		IF
			LEN(stMqttSettings.sMqttUserId) > 0
			AND LEN(stMqttSettings.sMqttPassword) > 0
		THEN
			iuLength := LEN(stMqttSettings.sMqttUserId)+2; (* 2 byte data length*)
			ipLength := LEN(stMqttSettings.sMqttPassword)+2; (* 2 byte data length*)
		ELSE
			iuLength := 0;
			ipLength := 0;
		END_IF

		(* Calculate length *)
		(* 10 byte header, 2 byte data length, data length, [user length + 2], [password length + 2]*)
		fbMqttEncodeLength(
			dwLength := 10 + 2 + INT_TO_BYTE(idLength) + INT_TO_BYTE(iuLength) + INT_TO_BYTE(ipLength),
			bLength1 => bLength1,
			bLength2 => bLength2,
			bLength3 => bLength3,
			bLength4 => bLength4,
			bAmount	 => bLengthAmount
		);

		(* MQTT Control Packet type *)
		stMqttTelegram.arMqttData[0] := 16;
		(* Remaining Length *)
		CASE bLengthAmount OF
			1:
				stMqttTelegram.arMqttData[1] := bLength1;

			2:
				stMqttTelegram.arMqttData[1] := bLength1;
				stMqttTelegram.arMqttData[2] := bLength2;

			3:
				stMqttTelegram.arMqttData[1] := bLength1;
				stMqttTelegram.arMqttData[2] := bLength2;
				stMqttTelegram.arMqttData[3] := bLength3;

			4:
				stMqttTelegram.arMqttData[1] := bLength1;
				stMqttTelegram.arMqttData[2] := bLength2;
				stMqttTelegram.arMqttData[3] := bLength3;
				stMqttTelegram.arMqttData[4] := bLength4;
		END_CASE;
		(* init position*)
		ipos := bLengthAmount;

		(* Length MSB *)
		stMqttTelegram.arMqttData[ipos+1] := 0;
		(* Length LSB *)
		stMqttTelegram.arMqttData[ipos+2] := 4;
		(* M *)
		stMqttTelegram.arMqttData[ipos+3] := 77;
		(* Q *)
		stMqttTelegram.arMqttData[ipos+4] := 81;
		(* T *)
		stMqttTelegram.arMqttData[ipos+5] := 84;
		(* T *)
		stMqttTelegram.arMqttData[ipos+6] := 84;
		(* Protocol Level *)
		stMqttTelegram.arMqttData[ipos+7] := 4;
		(* Connect Flags *)
		stMqttTelegram.arMqttData[ipos+8].1 := TRUE;
		stMqttTelegram.arMqttData[ipos+8].6 := (ipLength>2); (* more then 2 byte data length*)
		stMqttTelegram.arMqttData[ipos+8].7 := (iuLength>2); (* more then 2 byte data length*)
		(* Keep Alive MSB *)
		stMqttTelegram.arMqttData[ipos+9] := 0;
		(* Keep Alive LSB *)
		stMqttTelegram.arMqttData[ipos+10] := stMqttSettings.usKeepAliveTime;
		(* Data length MSB *)
		stMqttTelegram.arMqttData[ipos+11] := 0;
		(* Data length LSB *)
		stMqttTelegram.arMqttData[ipos+12] := INT_TO_BYTE(idLength);

		(* Client ID *)
		MEMCPY(
			destAddr	:= ADR(stMqttTelegram.arMqttData[ipos+13]),
		    srcAddr		:= ADR(stMqttSettings.sMqttClientId),
			n  			:= idLength
		);

		ipos := ipos+13+idLength;
		IF (iuLength > 2) THEN (* more then 2 byte data length*)
			(* Data length MSB *)
			stMqttTelegram.arMqttData[ipos] := 0;
			(* Data length LSB *)
			stMqttTelegram.arMqttData[ipos+1] := INT_TO_BYTE(iuLength-2);

			(* User ID *)
			MEMCPY(
				destAddr	:= ADR(stMqttTelegram.arMqttData[ipos+2]),
			    srcAddr		:= ADR(stMqttSettings.sMqttUserId),
				n  			:= iuLength-2
			);
			ipos := ipos+iuLength;
		END_IF

		IF (iuLength > 2) THEN (* more then 2 byte data length*)
			(* Data length MSB *)
			stMqttTelegram.arMqttData[ipos] := 0;
			(* Data length LSB *)
			stMqttTelegram.arMqttData[ipos+1] := INT_TO_BYTE(ipLength-2);

			(* Password *)
			MEMCPY(
				destAddr	:= ADR(stMqttTelegram.arMqttData[ipos+2]),
			    srcAddr		:= ADR(stMqttSettings.sMqttPassword),
				n  			:= ipLength-2
			);
			ipos := ipos+ipLength;
		END_IF

		stMqttTelegram.nDataLength 	:= ipos; (* 1 byte header, 1 byte remaining length *)
		iState 						:= C_SEND_WAIT;

	(* send telegram *)
	C_SEND_WAIT:
		IF stMqttSettings.stMqttSendTelegram.nDataLength = 0 THEN
			FC_Mqtt_CopyTelegram_V10(
				stMqttSrcTelegram	:= stMqttTelegram,
				stMqttDestTelegram	:= stMqttSettings.stMqttSendTelegram,
				stMqttSettings		:= stMqttSettings
			);

			stMqttSettings.bConnectPackageSent	:= TRUE;
			iState								:= C_IDLE;
		END_IF;

		IF
			NOT stMqttSettings.bActive
			OR NOT stMqttSettings.bSocketConnection
		THEN
			iState := C_STARTUP;
		END_IF;

	(* idle *)
	C_IDLE:
		IF
			NOT stMqttSettings.bDisconnect
			AND NOT stMqttSettings.bError
			AND NOT stMqttSettings.bConnected
			AND stMqttSettings.bSocketConnection
			AND NOT stMqttSettings.bConnectPackageSent
			AND stMqttSettings.bActive
		THEN
			iState := C_BUILD_CONNECT;
		END_IF;

		(* check received telegram *)
		IF
			stMqttSettings.bConnectPackageSent
			AND stMqttSettings.stMqttReceivedTelegram.nDataLength = 4
			AND stMqttSettings.stMqttReceivedTelegram.arMqttData[0] = 32
			AND stMqttSettings.stMqttReceivedTelegram.arMqttData[1] = 2
			AND (
				(* Session pressent or not, we ignore *)
				stMqttSettings.stMqttReceivedTelegram.arMqttData[2] = 1
				OR
				stMqttSettings.stMqttReceivedTelegram.arMqttData[2] = 0
			)
			AND stMqttSettings.stMqttReceivedTelegram.arMqttData[3] = 0
		THEN
			stMqttSettings.bConnected := TRUE;
			FC_Mqtt_ClearTelegram_V10(
				stMqttTelegram	:= stMqttSettings.stMqttReceivedTelegram,
				stMqttSettings	:= stMqttSettings
			);
		END_IF;

		(* error on connect *)
		IF
			stMqttSettings.bConnectPackageSent
			AND stMqttSettings.stMqttReceivedTelegram.nDataLength = 4
			AND stMqttSettings.stMqttReceivedTelegram.arMqttData[0] = 32
			AND stMqttSettings.stMqttReceivedTelegram.arMqttData[1] = 2
			AND stMqttSettings.stMqttReceivedTelegram.arMqttData[3] <> 0
		THEN
			stMqttSettings.bError := TRUE;
		END_IF;

		IF
			stMqttSettings.bDisconnect
			OR stMqttSettings.bError
			OR NOT stMqttSettings.bSocketConnection
			OR NOT stMqttSettings.bActive
		THEN
			iState := C_STARTUP;
		END_IF;

	ELSE
		iState := C_STARTUP;
END_CASE;


(*	END_FUNCTION_BLOCK	*)
END_FUNCTION_BLOCK

(* POU _Generic/Mqtt/Intern/FB_Mqtt_EncodeLength_V10, ST *)
FUNCTION_BLOCK FB_Mqtt_EncodeLength_V10
VAR_INPUT
	dwLength	: DWORD;
END_VAR
VAR_OUTPUT
	bLength1	: BYTE := 0;
	bLength2	: BYTE := 0;
	bLength3	: BYTE := 0;
	bLength4	: BYTE := 0;
	bAmount		: BYTE := 0;
END_VAR
VAR
	dwWorkLength	: DWORD;
	dwCopyLength	: DWORD;
END_VAR
(* @END_DECLARATION := '0' *)
bAmount 		:= 1;
dwCopyLength	:= dwLength;

WHILE dwCopyLength > 0 DO
	dwWorkLength := dwCopyLength MOD 128;
	dwCopyLength := dwCopyLength / 128;

	IF dwCopyLength > 0 THEN
		dwWorkLength := dwWorkLength OR 128;
	END_IF;

	CASE bAmount OF
		1:
			bLength1 := DWORD_TO_BYTE(dwWorkLength);

		2:
			bLength2 := DWORD_TO_BYTE(dwWorkLength);

		3:
			bLength3 := DWORD_TO_BYTE(dwWorkLength);

		4:
			bLength4 := DWORD_TO_BYTE(dwWorkLength);

		ELSE
			;
	END_CASE;

	IF dwCopyLength > 0 THEN
		bAmount := bAmount + 1;
	END_IF;

	IF bAmount > 4 THEN
		(* hmm *)
		RETURN;
	END_IF;
END_WHILE;
(*
do
	encodedByte = X MOD 128
	X = X DIV 128

	// if there are more data to encode, set the top bit of this byte
	if ( X > 0 )
		encodedByte = encodedByte OR 128
	endif

	'output' encodedByte
while ( X > 0 )
*)

(*	END_FUNCTION_BLOCK	*)
END_FUNCTION_BLOCK

(* POU _Generic/Mqtt/Intern/FC_Mqtt_ClearTelegram_V10, ST *)
FUNCTION FC_Mqtt_ClearTelegram_V10 : BOOL
VAR_IN_OUT
	stMqttTelegram	: ST_MqttTelegram;
	stMqttSettings	: ST_MqttSettings;
END_VAR
VAR
END_VAR
(* @END_DECLARATION := '0' *)
MEMSET(
	destAddr	:= ADR(stMqttTelegram.arMqttData),
	fillByte  	:= 0,
	n			:= stMqttSettings.iTelegramSize
);

stMqttTelegram.nDataLength := 0;

(*	END_FUNCTION	*)
END_FUNCTION

(* POU _Generic/Mqtt/Intern/FC_Mqtt_CopyTelegram_V10, ST *)
FUNCTION FC_Mqtt_CopyTelegram_V10 : BOOL
VAR_IN_OUT
	stMqttSrcTelegram	: ST_MqttTelegram;
	stMqttDestTelegram	: ST_MqttTelegram;
	stMqttSettings		: ST_MqttSettings;
END_VAR
VAR
END_VAR
(* @END_DECLARATION := '0' *)
MEMCPY(
	destAddr	:= ADR(stMqttDestTelegram.arMqttData),
    srcAddr		:= ADR(stMqttSrcTelegram.arMqttData),
	n  			:= stMqttSettings.iTelegramSize
);

stMqttDestTelegram.nDataLength := stMqttSrcTelegram.nDataLength;

(*	END_FUNCTION	*)
END_FUNCTION

(* POU _Generic/Mqtt/Intern/FB_MqttTelegram_PingReq_V10, ST *)
FUNCTION_BLOCK FB_MqttTelegram_PingReq_V10
VAR_IN_OUT
	stMqttSettings	: ST_MqttSettings;
END_VAR
VAR
	iState 				: INT := 0;
	bMustSend			: BOOL := FALSE;
	bPingReqSent		: BOOL := FALSE;
	stMqttTelegram		: ST_MqttTelegram;
END_VAR
VAR CONSTANT
	C_STARTUP		: INT := 0;
	C_BUILD_PING	: INT := 100;
	C_SEND_WAIT		: INT := 110;
	C_IDLE			: INT := 500;
END_VAR
(* @END_DECLARATION := '0' *)
CASE iState OF
	C_STARTUP:
		bPingReqSent := FALSE;

		IF stMqttSettings.bValidConnection THEN
			iState := C_IDLE;
		END_IF;

	(* build pingreq telegram *)
	C_BUILD_PING:
		FC_Mqtt_ClearTelegram_V10(
			stMqttTelegram	:= stMqttTelegram,
			stMqttSettings	:= stMqttSettings
		);

		(* MQTT Control Packet type *)
		stMqttTelegram.arMqttData[0] := 192;
		(* Remaining Length *)
		stMqttTelegram.arMqttData[1] := 0;

		stMqttTelegram.nDataLength := 2;

		iState := C_SEND_WAIT;

	(* send telegram *)
	C_SEND_WAIT:
		IF stMqttSettings.stMqttSendTelegram.nDataLength = 0 THEN
			FC_Mqtt_CopyTelegram_V10(
				stMqttSrcTelegram	:= stMqttTelegram,
				stMqttDestTelegram	:= stMqttSettings.stMqttSendTelegram,
				stMqttSettings		:= stMqttSettings
			);

			bPingReqSent	:= TRUE;
			iState			:= C_IDLE;
		END_IF;

		IF NOT stMqttSettings.bValidConnection THEN
			iState := C_STARTUP;
		END_IF;

	(* idle *)
	C_IDLE:
		bMustSend := FALSE;

		IF stMqttSettings.usKeepAliveTime > 0 THEN
			bMustSend := stMqttSettings.tonSendPingReq.Q;
		END_IF;

		IF
			stMqttSettings.bValidConnection
			AND bMustSend
			AND NOT bPingReqSent
		THEN
			iState := C_BUILD_PING;
		END_IF;

		(* Check received telegram *)
		IF
			bPingReqSent
			AND stMqttSettings.stMqttReceivedTelegram.nDataLength = 2
			AND stMqttSettings.stMqttReceivedTelegram.arMqttData[0] = 208
			AND stMqttSettings.stMqttReceivedTelegram.arMqttData[1] = 0
		THEN
			FC_Mqtt_ClearTelegram_V10(
				stMqttTelegram	:= stMqttSettings.stMqttReceivedTelegram,
				stMqttSettings	:= stMqttSettings
			);
			bPingReqSent := FALSE;
		END_IF;

		IF NOT stMqttSettings.bValidConnection THEN
			iState := C_STARTUP;
		END_IF;

	ELSE
		iState := C_STARTUP;
END_CASE;

(*	END_FUNCTION_BLOCK	*)
END_FUNCTION_BLOCK

(* POU _Generic/Mqtt/Intern/FB_Mqtt_Send_V10, ST *)
FUNCTION_BLOCK FB_Mqtt_Send_V10
VAR_OUTPUT
	bBusy	: BOOL := FALSE;
END_VAR
VAR_IN_OUT
	stMqttSettings	: ST_MqttSettings;
END_VAR
VAR
	fbSocketSend 	: FB_SocketSend;
	tPingReq		: TIME;
	iState 			: INT := 0;
	stSendTelegram	: ST_MqttTelegram;
END_VAR
VAR CONSTANT
	C_STARTUP		: INT := 0;
	C_SEND			: INT := 100;
	C_SEND_WAIT		: INT := 110;
	C_IDLE			: INT := 500;
END_VAR
(* @END_DECLARATION := '0' *)
CASE iState OF
	C_STARTUP:
		bBusy := FALSE;

		stMqttSettings.tonSendPingReq(
			in := FALSE
		);

		IF
			NOT stMqttSettings.bDisconnect
			AND NOT stMqttSettings.bError
			AND stMqttSettings.bSocketConnection
		THEN
			iState := C_IDLE;
		END_IF;

	(* send mqtt telegram *)
	C_SEND:
		bBusy := TRUE;

		(* copy send telegram *)
		FC_Mqtt_CopyTelegram_V10(
			stMqttSrcTelegram	:= stMqttSettings.stMqttSendTelegram,
			stMqttDestTelegram	:= stSendTelegram,
			stMqttSettings		:= stMqttSettings
		);

		(* start send *)
		fbSocketSend(
			bExecute := FALSE
		);

		fbSocketSend(
			sSrvNetId	:= '',
			hSocket		:= stMqttSettings.hSocket,
			cbLen		:= stSendTelegram.nDataLength,
			pSrc		:= ADR(stSendTelegram.arMqttData),
			bExecute 	:= TRUE
		);

		iState := C_SEND_WAIT;

	(* wait send done *)
	C_SEND_WAIT:
		fbSocketSend(
			bExecute := FALSE
		);

		IF
			NOT fbSocketSend.bBusy
			AND NOT fbSocketSend.bError
		THEN
			(* copy last telegram *)
			FC_Mqtt_CopyTelegram_V10(
				stMqttSrcTelegram	:= stMqttSettings.stMqttSendTelegram,
				stMqttDestTelegram	:= stMqttSettings.stMqttLastSendTelegram,
				stMqttSettings		:= stMqttSettings
			);

			(* clear send buffer *)
			FC_Mqtt_ClearTelegram_V10(
				stMqttTelegram 	:= stMqttSettings.stMqttSendTelegram,
				stMqttSettings	:= stMqttSettings
			);

			iState	:= C_IDLE;
			bBusy	:= FALSE;
		END_IF;

		IF stMqttSettings.usKeepAliveTime > 0 THEN
			tPingReq := DWORD_TO_TIME(USINT_TO_DWORD(stMqttSettings.usKeepAliveTime) * 1000 - 5000);

			stMqttSettings.tonSendPingReq(
				in := FALSE
			);

			stMqttSettings.tonSendPingReq(
				in := TRUE,
				pt := tPingReq
			);
		END_IF;

		IF fbSocketSend.bError THEN
			iState 					:= C_STARTUP;
			stMqttSettings.bError	:= TRUE;
		END_IF;

		IF
			NOT stMqttSettings.bActive
			OR NOT stMqttSettings.bSocketConnection
		THEN
			iState := C_STARTUP;
		END_IF;

	(* idle *)
	C_IDLE:
		IF stMqttSettings.usKeepAliveTime > 0 THEN
			stMqttSettings.tonSendPingReq(
				in := stMqttSettings.bConnected
			);
		ELSE
			stMqttSettings.tonSendPingReq(
				in := FALSE
			);
		END_IF;

		IF
			stMqttSettings.stMqttSendTelegram.nDataLength > 0
			AND NOT stMqttSettings.bDisconnect
			AND NOT stMqttSettings.bError
			AND stMqttSettings.bSocketConnection
			AND NOT bBusy
		THEN
			iState := C_SEND;
		END_IF;

		IF
			stMqttSettings.bDisconnect
			OR stMqttSettings.bError
			OR NOT stMqttSettings.bSocketConnection
		THEN
			iState := C_STARTUP;
		END_IF;

		(* ensure at least 1 cycle pause *)
		(* bBusy := FALSE; *)

	ELSE
		iState := C_STARTUP;
END_CASE;

(*	END_FUNCTION_BLOCK	*)
END_FUNCTION_BLOCK

(* POU _Generic/Mqtt/Intern/FB_Mqtt_Receive_V10, ST *)
FUNCTION_BLOCK FB_Mqtt_Receive_V10
VAR_OUTPUT
	bBusy	: BOOL := FALSE;
END_VAR
VAR_IN_OUT
	stMqttSettings	: ST_MqttSettings;
END_VAR
VAR
	fbSocketReceive		: FB_SocketReceive;
	fbMqttDecodeLength	: FB_Mqtt_DecodeLength_V10;
	stReceiveBuffer		: ST_MqttTelegram;

	iState 			: INT := 0;
	iLengthPosition	: INT := 0;
	index			: INT := 0;
	dwDataLength	: DWORD := 0;
	wTopicLength	: WORD := 0;
	dwValueLength	: DWORD := 0;
END_VAR
VAR CONSTANT
	C_STARTUP				: INT := 0;
	C_RECEIVE_HEADER		: INT := 100;
	C_RECEIVE_HEADER_WAIT	: INT := 110;
	C_RECEIVE_LENGTH		: INT := 120;
	C_RECEIVE_LENGTH_WAIT	: INT := 130;
	C_RECEIVE_DATA			: INT := 200;
	C_RECEIVE_DATA_WAIT		: INT := 210;
	C_IDLE					: INT := 500;
END_VAR
(* @END_DECLARATION := '0' *)
CASE iState OF
	C_STARTUP:
		bBusy 			:= FALSE;
		iLengthPosition	:= 0;
		index			:= 0;
		dwDataLength	:= 0;
		wTopicLength	:= 0;
		dwValueLength	:= 0;
		ClearReceivedPublishTelegram();

		IF
			NOT stMqttSettings.bDisconnect
			AND NOT stMqttSettings.bError
			AND stMqttSettings.bSocketConnection
		THEN
			iState := C_IDLE;
		END_IF;

	(* start receive header *)
	C_RECEIVE_HEADER:
		bBusy := TRUE;
		ClearReceivedPublishTelegram();

		fbSocketReceive(
			bExecute := FALSE
		);

		fbSocketReceive(
			sSrvNetId	:= '',
			hSocket		:= stMqttSettings.hSocket,
			cbLen		:= 2,
			pDest		:= ADR(stReceiveBuffer.arMqttData),
			bExecute 	:= TRUE
		);

		iState := C_RECEIVE_HEADER_WAIT;

	(* wait for header with length *)
	C_RECEIVE_HEADER_WAIT:
		fbSocketReceive(
			bExecute := FALSE
		);

		IF
			NOT fbSocketReceive.bBusy
			AND NOT fbSocketReceive.bError
			AND fbSocketReceive.nRecBytes = 2
		THEN
			iLengthPosition	:= 0;
			stMqttSettings.stMqttReceivedTelegram.arMqttData[0] := stReceiveBuffer.arMqttData[0];
			stMqttSettings.stMqttReceivedTelegram.arMqttData[1] := stReceiveBuffer.arMqttData[1];

			IF stMqttSettings.stMqttReceivedTelegram.arMqttData[1].7 = 1 THEN
				(* payload longer then 127 byte *)
				iLengthPosition := iLengthPosition + 1;
				iState			:= C_RECEIVE_LENGTH;
			ELSE
				IF stMqttSettings.stMqttReceivedTelegram.arMqttData[1] = 0 THEN
					(* no payload received *)
					stMqttSettings.stMqttReceivedTelegram.nDataLength := 2;

					(* copy last telegram *)
					FC_Mqtt_CopyTelegram_V10(
						stMqttSrcTelegram	:= stMqttSettings.stMqttReceivedTelegram,
						stMqttDestTelegram	:= stMqttSettings.stMqttLastReceivedTelegram,
						stMqttSettings		:= stMqttSettings
					);

					iState	:= C_IDLE;
					bBusy 	:= FALSE;
				ELSE
					iState := C_RECEIVE_DATA;
				END_IF;
			END_IF;
		END_IF;

		IF fbSocketReceive.bError THEN
			iState 					:= C_STARTUP;
			stMqttSettings.bError	:= TRUE;
		END_IF;

		IF fbSocketReceive.nRecBytes = 0 THEN
			iState	:= C_IDLE;
			bBusy	:= FALSE;
		END_IF;

		IF
			NOT stMqttSettings.bActive
			OR NOT stMqttSettings.bSocketConnection
		THEN
			iState := C_STARTUP;
		END_IF;

	(* read next remaining length *)
	C_RECEIVE_LENGTH:
		fbSocketReceive(
			bExecute := FALSE
		);

		fbSocketReceive(
			sSrvNetId	:= '',
			hSocket		:= stMqttSettings.hSocket,
			cbLen		:= 1,
			pDest		:= ADR(stReceiveBuffer.arMqttData),
			bExecute 	:= TRUE
		);

		iState := C_RECEIVE_LENGTH_WAIT;

	(* wait for remaining length *)
	C_RECEIVE_LENGTH_WAIT:
		fbSocketReceive(
			bExecute := FALSE
		);

		IF
			NOT fbSocketReceive.bBusy
			AND NOT fbSocketReceive.bError
			AND fbSocketReceive.nRecBytes = 1
		THEN
			stMqttSettings.stMqttReceivedTelegram.arMqttData[1 + iLengthPosition] := stReceiveBuffer.arMqttData[0];

			IF stMqttSettings.stMqttReceivedTelegram.arMqttData[1 + iLengthPosition].7 = 1 THEN
				(* read next length byte *)
				iLengthPosition := iLengthPosition + 1;
				iState			:= C_RECEIVE_LENGTH;

				(* Not more the 4 length bytes *)
				IF iLengthPosition > 4 THEN
					iState 					:= C_STARTUP;
					stMqttSettings.bError	:= TRUE;
				END_IF;
			ELSE
				iState := C_RECEIVE_DATA;
			END_IF;
		END_IF;

		IF fbSocketReceive.bError THEN
			iState 					:= C_STARTUP;
			stMqttSettings.bError	:= TRUE;
		END_IF;

		IF
			NOT stMqttSettings.bActive
			OR NOT stMqttSettings.bSocketConnection
		THEN
			iState := C_STARTUP;
		END_IF;

	(* receive remaining data *)
	C_RECEIVE_DATA:
		fbMqttDecodeLength(
			stMqttTelegram	:= stMqttSettings.stMqttReceivedTelegram,
			dwLength		=> dwDataLength
		);

		fbSocketReceive(
			bExecute := FALSE
		);

		fbSocketReceive(
			sSrvNetId	:= '',
			hSocket		:= stMqttSettings.hSocket,
			cbLen		:= dwDataLength,
			pDest		:= ADR(stReceiveBuffer.arMqttData),
			bExecute 	:= TRUE
		);

		iState := C_RECEIVE_DATA_WAIT;

	(* receive *)
	C_RECEIVE_DATA_WAIT:
		fbSocketReceive(
			bExecute := FALSE
		);

		IF
			NOT fbSocketReceive.bBusy
			AND NOT fbSocketReceive.bError
			AND fbSocketReceive.nRecBytes > 0
		THEN
			MEMCPY(
				destAddr	:= ADR(stMqttSettings.stMqttReceivedTelegram.arMqttData[2 + iLengthPosition]),
			    srcAddr		:= ADR(stReceiveBuffer.arMqttData),
				n  			:= fbSocketReceive.nRecBytes
			);
			stMqttSettings.stMqttReceivedTelegram.nDataLength := 2 + iLengthPosition + fbSocketReceive.nRecBytes;

			(* copy last telegram *)
			FC_Mqtt_CopyTelegram_V10(
				stMqttSrcTelegram	:= stMqttSettings.stMqttReceivedTelegram,
				stMqttDestTelegram	:= stMqttSettings.stMqttLastReceivedTelegram,
				stMqttSettings		:= stMqttSettings
			);

			(* check for publish *)
			IF (stMqttSettings.stMqttReceivedTelegram.arMqttData[0] AND 48) = 48 THEN
				ClearReceivedPublishTelegram();

				(* Length MSB/LSB Topic *)
				wTopicLength :=
						SHL(BYTE_TO_WORD(stMqttSettings.stMqttReceivedTelegram.arMqttData[2 + iLengthPosition + 1]), 8) +
						BYTE_TO_WORD(stMqttSettings.stMqttReceivedTelegram.arMqttData[1 + iLengthPosition + 1]);
				wTopicLength := BE16_TO_HOST(wTopicLength);

				(* Copy topic *)
				MEMCPY(
					destAddr	:= ADR(stMqttSettings.stMqttReceivedPublishTelegram.sTopic),
				    srcAddr		:= ADR(stMqttSettings.stMqttReceivedTelegram.arMqttData[3 + iLengthPosition + 1]),
					n  			:= wTopicLength
				);

				(* Copy value *)
				(* value length = remaining data length - length topic value - 2 byte topic length *)
				dwValueLength := dwDataLength - wTopicLength - 2;

				MEMCPY(
					destAddr	:= ADR(stMqttSettings.stMqttReceivedPublishTelegram.sValue),
				    srcAddr		:= ADR(stMqttSettings.stMqttReceivedTelegram.arMqttData[3 + iLengthPosition + 1 + wTopicLength]),
					n  			:= dwValueLength
				);

				stMqttSettings.stMqttReceivedPublishTelegram.bHasData := TRUE;
			END_IF;

			iState	:= C_IDLE;
			bBusy	:= FALSE;
		END_IF;

		IF fbSocketReceive.bError THEN
			iState 					:= C_STARTUP;
			stMqttSettings.bError	:= TRUE;
		END_IF;

		IF
			NOT stMqttSettings.bActive
			OR NOT stMqttSettings.bSocketConnection
		THEN
			iState := C_STARTUP;
		END_IF;

	(* idle *)
	C_IDLE:
		IF
			NOT stMqttSettings.bDisconnect
			AND NOT stMqttSettings.bError
			AND stMqttSettings.bSocketConnection
			AND NOT bBusy
		THEN
			iState := C_RECEIVE_HEADER;
		END_IF;

		IF
			stMqttSettings.bDisconnect
			OR stMqttSettings.bError
			OR NOT stMqttSettings.bSocketConnection
		THEN
			iState := C_STARTUP;
		END_IF;

		(* ensure at least 1 cycle pause *)
		(* bBusy := FALSE; *)

	ELSE
		iState := C_STARTUP;
END_CASE;

(*	END_FUNCTION_BLOCK	*)
END_FUNCTION_BLOCK
ACTION ClearReceivedPublishTelegram:
MEMSET(
	destAddr	:= ADR(stMqttSettings.stMqttReceivedPublishTelegram.sTopic),
	fillByte  	:= 0,
	n			:= 255
);
stMqttSettings.stMqttReceivedPublishTelegram.sTopic := '';

MEMSET(
	destAddr	:= ADR(stMqttSettings.stMqttReceivedPublishTelegram.sValue),
	fillByte  	:= 0,
	n			:= 255
);
stMqttSettings.stMqttReceivedPublishTelegram.sValue := '';

stMqttSettings.stMqttReceivedPublishTelegram.bHasData := FALSE;
END_ACTION

(* POU _Generic/Mqtt/Intern/FB_Mqtt_DecodeLength_V10, ST *)
FUNCTION_BLOCK FB_Mqtt_DecodeLength_V10
VAR_INPUT
	stMqttTelegram : ST_MqttTelegram;
END_VAR
VAR_OUTPUT
	dwLength	: DWORD;
	bAmount		: BYTE;
END_VAR
VAR
	index			: INT;
	diMultiplier	: DINT;
	dwValue			: DWORD;
END_VAR
(* @END_DECLARATION := '0' *)
index			:= 0;
diMultiplier	:= 1;
dwValue			:= 0;

REPEAT
	index := index + 1;

	dwValue := dwValue + (stMqttTelegram.arMqttData[index] AND 127) * diMultiplier;
	diMultiplier := diMultiplier * 128;

	IF diMultiplier > 128*128*128 THEN
		dwLength	:= 0;
		bAmount		:= 0;
		RETURN;
	END_IF;
UNTIL stMqttTelegram.arMqttData[index].7 = 0
END_REPEAT;

dwLength	:= dwValue;
bAmount		:= INT_TO_BYTE(index);

(*
multiplier = 1
value = 0

do
	encodedByte = 'next byte from stream'
	value += (encodedByte AND 127) * multiplier
	multiplier *= 128

	if (multiplier > 128*128*128)
		throw Error(Malformed Remaining Length)
while ((encodedByte AND 128) != 0)

*)

(*	END_FUNCTION_BLOCK	*)
END_FUNCTION_BLOCK

(* POU _Generic/Mqtt/FB_Mqtt_Publish_V10, ST *)
FUNCTION_BLOCK FB_Mqtt_Publish_V10
VAR_INPUT
	sTopic	: STRING[255];
	sValue	: STRING[255];
	bRetain	: BOOL := TRUE;
END_VAR
VAR_OUTPUT
	bBusy	: BOOL := FALSE;
END_VAR
VAR_IN_OUT
	stMqttSettings	: ST_MqttSettings;
END_VAR
VAR
	bFirstPublishDone	: BOOL := FALSE;
	bMustPublish		: BOOL := FALSE;
	sLastValue			: STRING[255];
	iState 				: INT := 0;
	iLengthTopic		: INT := 0;
	iLengthValue		: INT := 0;
	wTopicLength		: WORD;
	stMqttTelegram		: ST_MqttTelegram;
	fbMqttEncodeLength	: FB_Mqtt_EncodeLength_V10;
	bLength1			: BYTE;
	bLength2			: BYTE;
	bLength3			: BYTE;
	bLength4			: BYTE;
	bLengthAmount		: BYTE;
END_VAR
VAR CONSTANT
	C_STARTUP			: INT := 0;
	C_BUILD_TELEGRAM	: INT := 100;
	C_SEND_WAIT			: INT := 110;
	C_IDLE				: INT := 500;
END_VAR
(* @END_DECLARATION := '0' *)
CASE iState OF
	C_STARTUP:
		bFirstPublishDone	:= FALSE;
		bBusy				:= FALSE;

		IF stMqttSettings.bValidConnection THEN
			iState := C_IDLE;
		END_IF;

	(* build publish telegram *)
	C_BUILD_TELEGRAM:
		bBusy := TRUE;
		iLengthTopic := LEN(sTopic);
		iLengthValue := LEN(sValue);

		FC_Mqtt_ClearTelegram_V10(
			stMqttTelegram	:= stMqttTelegram,
			stMqttSettings	:= stMqttSettings
		);

		wTopicLength := iLengthTopic;
		wTopicLength := HOST_TO_BE16(wTopicLength);

		(* Calculate length *)
		(* 2 byte length topic, x byte length topic, x byte length value *)
		fbMqttEncodeLength(
			dwLength := 2 + iLengthTopic + iLengthValue,
			bLength1 => bLength1,
			bLength2 => bLength2,
			bLength3 => bLength3,
			bLength4 => bLength4,
			bAmount	 => bLengthAmount
		);

		(* MQTT Control Packet type, no DUP, no QoS, Retain *)
		stMqttTelegram.arMqttData[0] := 48;
		IF bRetain THEN
			stMqttTelegram.arMqttData[0].0 := 1;
		END_IF;

		(* Remaining Length *)
		CASE bLengthAmount OF
			1:
				stMqttTelegram.arMqttData[1] := bLength1;

			2:
				stMqttTelegram.arMqttData[1] := bLength1;
				stMqttTelegram.arMqttData[2] := bLength2;

			3:
				stMqttTelegram.arMqttData[1] := bLength1;
				stMqttTelegram.arMqttData[2] := bLength2;
				stMqttTelegram.arMqttData[3] := bLength3;

			4:
				stMqttTelegram.arMqttData[1] := bLength1;
				stMqttTelegram.arMqttData[2] := bLength2;
				stMqttTelegram.arMqttData[3] := bLength3;
				stMqttTelegram.arMqttData[4] := bLength4;

			ELSE
				iState 					:= C_STARTUP;
				stMqttSettings.bError	:= TRUE;
		END_CASE;

		(* Length MSB Topic *)
		stMqttTelegram.arMqttData[1 + bLengthAmount] := WORD_TO_BYTE(wTopicLength);
		(* Length LSB Topic *)
		stMqttTelegram.arMqttData[2 + bLengthAmount] := WORD_TO_BYTE(SHR(wTopicLength, 8));

		(* Add topic *)
		MEMCPY(
			destAddr	:= ADR(stMqttTelegram.arMqttData[3 + bLengthAmount]),
		    srcAddr		:= ADR(sTopic),
			n  			:= iLengthTopic
		);

		(* Add Payload *)
		MEMCPY(
			destAddr	:= ADR(stMqttTelegram.arMqttData[3 + bLengthAmount + iLengthTopic]),
		    srcAddr		:= ADR(sValue),
			n  			:= iLengthValue
		);

		(* 1 byte header, x byte variable length, 2 byte topic lenght, x byte topic, x byte value *)
		stMqttTelegram.nDataLength := 1 + bLengthAmount + 2 + iLengthTopic + iLengthValue;

		iState := C_SEND_WAIT;

	(* send telegram *)
	C_SEND_WAIT:
		IF stMqttSettings.stMqttSendTelegram.nDataLength = 0 THEN
			FC_Mqtt_CopyTelegram_V10(
				stMqttSrcTelegram	:= stMqttTelegram,
				stMqttDestTelegram	:= stMqttSettings.stMqttSendTelegram,
				stMqttSettings		:= stMqttSettings
			);

			iState				:= C_IDLE;
			bFirstPublishDone	:= TRUE;
			sLastValue			:= sValue;
		END_IF;

		IF NOT stMqttSettings.bValidConnection THEN
			iState := C_STARTUP;
		END_IF;

	(* idle *)
	C_IDLE:
		bBusy 			:= FALSE;
		bMustPublish 	:= sLastValue <> sValue;

		IF
			stMqttSettings.bValidConnection
			AND (
				bMustPublish
				OR NOT bFirstPublishDone
			)
		THEN
			iState := C_BUILD_TELEGRAM;
		END_IF;

		IF NOT stMqttSettings.bValidConnection THEN
			iState := C_STARTUP;
		END_IF;

	ELSE
		iState := C_STARTUP;
END_CASE;

(*	END_FUNCTION_BLOCK	*)
END_FUNCTION_BLOCK

(* POU ParnikWindowCtrl_old, ST *)
PROGRAM ParnikWindowCtrl_old
VAR
    (* Modbus I/O (использовать точно как заданы) *)
    (* Modbus.Street_temp : REAL *)
    (* Modbus.Parnik_set_temp_street_min : REAL *)
    (* Modbus.Parnik_air_temp : REAL *)
    (* Modbus.Parnik_set_auto_window : BOOL *)
    (* Modbus.Parnik_current_level_window : UINT *) (* 0=closed,1=30%,2=60%,3=100% *)
    (* Modbus.Parnik_manual_level_window : UINT *)
    (* Modbus.Parnik_temp_step1_window : UINT *) (* threshold for 30% *)
    (* Modbus.Parnik_temp_step2_window : UINT *) (* threshold for 60% *)

    (* HW outputs *)
    (* HW_power_supply_parnik : BOOL *)
    (* HW_power_polarity_parnik : BOOL *)

    (* Internal *)
    closeTON : TON;                 (* PT = 60s *)
    openTON  : TON;                 (* PT = variable *)
    state : UINT := 0;              (* 0=idle,1=closing,2=opening *)
    targetLevel : UINT := 0;        (* desired final level 0..3 *)
    openTime : TIME := T#0s;
    hysteresis : REAL := 4.0;
    prevManualLevel : UINT := 255;
    manualReq : BOOL := FALSE;
    startClose : BOOL := FALSE;
    startOpen  : BOOL := FALSE;
    firstScan : BOOL := TRUE;
END_VAR
IF firstScan THEN
    Modbus.Parnik_current_level_window := 0; (* default closed *)
    HW_power_supply_parnik := FALSE;
    HW_power_polarity_parnik := FALSE;
    closeTON(IN := FALSE, PT := T#60s);
    openTON(IN := FALSE, PT := T#60s);
    prevManualLevel := Modbus.Parnik_manual_level_window;
    firstScan := FALSE;
END_IF

(* detect manual change request *)
manualReq := FALSE;
IF NOT Modbus.Parnik_set_auto_window THEN
    IF Modbus.Parnik_manual_level_window <> prevManualLevel THEN
        manualReq := TRUE;
    END_IF;
END_IF;
prevManualLevel := Modbus.Parnik_manual_level_window;

(* Determine targetLevel according to requested logic *)
IF Modbus.Parnik_set_auto_window THEN
    (* AUTO *)
    IF (Modbus.Parnik_air_temp > (INT_TO_REAL(Modbus.Parnik_temp_step1_window) + hysteresis))
       AND (Modbus.Parnik_air_temp < INT_TO_REAL(Modbus.Parnik_temp_step2_window))
       AND (Modbus.Street_temp > Modbus.Parnik_set_temp_street_min) THEN
        targetLevel := 1; (* 30% *)
    ELSIF (Modbus.Parnik_air_temp > (INT_TO_REAL(Modbus.Parnik_temp_step2_window) + hysteresis))
       AND (Modbus.Street_temp > Modbus.Parnik_set_temp_street_min) THEN
        targetLevel := 2; (* 60% *)
    ELSIF ( (Modbus.Parnik_air_temp < (INT_TO_REAL(Modbus.Parnik_temp_step1_window) - hysteresis))
            OR (Modbus.Street_temp < Modbus.Parnik_set_temp_street_min) ) THEN
        targetLevel := 0; (* close *)
    ELSE
        targetLevel := Modbus.Parnik_current_level_window; (* keep current *)
    END_IF;
ELSE
    (* MANUAL - independent от температуры *)
    CASE Modbus.Parnik_manual_level_window OF
        0: targetLevel := 0;
        1: targetLevel := 1;
        2: targetLevel := 2;
        3: targetLevel := 3;
        ELSE targetLevel := Modbus.Parnik_current_level_window;
    END_CASE;
END_IF;


(* Helper: request sequence when target differs or when manualReq *)
IF state = 0 THEN
    startClose := FALSE;
    startOpen := FALSE;
    (* If target equals current -> nothing *)
    IF Modbus.Parnik_current_level_window <> targetLevel THEN
        IF targetLevel = 0 THEN
            (* need close *)
            startClose := TRUE;
            state := 1;
            HW_power_polarity_parnik := FALSE; (* closing polarity *)
        ELSE
            (* target > 0 *)
            IF Modbus.Parnik_current_level_window < targetLevel THEN
                (* already closed -> open directly *)
(*                IF openTime > T#0s THEN *)
                    startOpen := TRUE;
			IF (Modbus.Parnik_current_level_window = 0 AND targetLevel  = 1) THEN
		 	   openTime := T#5s;
			 END_IF
			IF (Modbus.Parnik_current_level_window = 0 AND targetLevel =  2) THEN
		 	   openTime := T#30s;
			 END_IF
			IF (Modbus.Parnik_current_level_window = 0 AND targetLevel =  3) THEN
		 	   openTime := T#60s;
			 END_IF
			IF (Modbus.Parnik_current_level_window = 1 AND targetLevel =  2) THEN
		 	   openTime := T#20s;
			 END_IF
			IF (Modbus.Parnik_current_level_window = 1 AND targetLevel =  3) THEN
		 	   openTime := T#50s;
			 END_IF
			IF (Modbus.Parnik_current_level_window = 2 AND targetLevel =  3) THEN
		 	   openTime := T#30s;
			 END_IF
                    state := 2;
                    HW_power_polarity_parnik := TRUE; (* opening polarity *)
            ELSE
                (* not closed -> close first *)
                startClose := TRUE;
                state := 1;
                HW_power_polarity_parnik := FALSE;
            END_IF;
        END_IF;
    END_IF;
END_IF

(* Also handle explicit manual request forcing sequence even if target==current but user changed set *)
IF manualReq AND (state = 0) THEN
    IF Modbus.Parnik_current_level_window <> targetLevel THEN
        (* same logic as above: if target>0 and already closed -> open; else close first *)
        IF targetLevel = 0 THEN
            startClose := TRUE; state := 1; HW_power_polarity_parnik := FALSE;
        ELSE
            IF Modbus.Parnik_current_level_window = 0 THEN
                IF openTime > T#0s THEN startOpen := TRUE; state := 2; HW_power_polarity_parnik := TRUE;
                ELSE Modbus.Parnik_current_level_window := targetLevel; state := 0;
                END_IF;
            ELSE
                startClose := TRUE; state := 1; HW_power_polarity_parnik := FALSE;
            END_IF;
        END_IF;
    END_IF;
END_IF

(* State machine with explicit TON IN handling *)
CASE state OF
    0: (* idle *)
        HW_power_supply_parnik := FALSE;
    1: (* closing - use full close time 60s *)
        closeTON(IN := startClose, PT := T#60s);
        HW_power_polarity_parnik := FALSE;
        HW_power_supply_parnik := startClose;

        IF closeTON.Q THEN
            (* finished closing *)
            closeTON(IN := FALSE, PT := T#60s);
            startClose := FALSE;
            HW_power_supply_parnik := FALSE;
            Modbus.Parnik_current_level_window := 0;
            (* If target >0 -> open to required level *)
            IF targetLevel > 0 THEN
                IF openTime > T#0s THEN
                    startOpen := TRUE;
                    state := 2;
                    HW_power_polarity_parnik := TRUE;
                ELSE
                    Modbus.Parnik_current_level_window := targetLevel;
                    state := 0;
                END_IF;
            ELSE
                state := 0;
            END_IF;
        END_IF;

    2: (* opening *)
        IF openTime = T#0s THEN
            startOpen := FALSE;
            HW_power_supply_parnik := FALSE;
            Modbus.Parnik_current_level_window := targetLevel;
            state := 0;
        ELSE
            openTON(IN := startOpen, PT := openTime);
            HW_power_polarity_parnik := TRUE;
            HW_power_supply_parnik := startOpen;

            IF openTON.Q THEN
                openTON(IN := FALSE, PT := openTime);
                startOpen := FALSE;
                HW_power_supply_parnik := FALSE;
                Modbus.Parnik_current_level_window := targetLevel;
                state := 0;
            END_IF;
        END_IF;

ELSE
    (* fallback safe *)
    HW_power_supply_parnik := FALSE;
    startClose := FALSE;
    startOpen := FALSE;
    closeTON(IN := FALSE, PT := T#60s);
    openTON(IN := FALSE, PT := openTime);
    state := 0;
END_CASE;
END_PROGRAM

(* POU RS485read_2_old, ST *)
PROGRAM RS485read_2_old
VAR
	password_1				: ARRAY [1..6] OF BYTE:=6(1); (* пароль к меркуриям, по умолчанию 6 единиц*)






	get_energy_E_T1			: FB_GET_ENERGY;
	get_energy_E_T2			: FB_GET_ENERGY;
	get_energy_MT			: FB_GET_ENERGY;
	get_supply				: FB_GET_SUPPLY;
	get_current				: FB_GET_CURRENT;
	get_power				: FB_GET_POWER;
	energyMT					: ARRAY[1..12,1..2] OF REAL;

	get_current_done			: BOOL;
	get_power_done			: BOOL;

	get_energy_E_T1_done	: BOOL;
	get_energy_E_T2_done	: BOOL;
	get_energy_MT_done		: BOOL;

	get_supply_done			: BOOL;
(*	CounterError_M			: DINT;
	CounterSuccess_M		: DINT;
*)




	flag: BOOL := TRUE;
	KLConfiguration: KL6configuration;
(*	Period_vent_switch	: INT:=180; *)
	CO2_period			: TIME;
	tTimerValue			: TIME	:=	t#10s; (* Период опроса RS485*)

	crctest					: WORD;

	arrReceive				: ARRAY[1..5] OF BYTE;
	arrSend					: ARRAY[1..5] OF BYTE;

	MBdata					 : ARRAY [1..2] OF INT;
	MBdata_pzem			 : ARRAY [1..2] OF INT;
	MBdata8					 : ARRAY [1..8] OF INT;
	FtrigBusy				: F_TRIG;
	timeoutvalue				: TIME := T#2000ms;		(* timeout while waiting for an answer of the modbus slave *)
	state					: INT;
	busy					: BOOL;
	LastErrorstate				: INT;
	LastModbusError			: ST_ModbusErrorDiagnostics;
	CounterError				: DINT;
	CounterSuccess			: DINT;

	i,k,l,m,t					: INT:=1;



	sensors_CO2_id				: ARRAY[1..2] OF BYTE:=16#68, 16#69;
	sensors_CO2_ppm			: ARRAY[1..2] OF INT;

	sensors_PZEM_id			: BYTE:=16#02;
	sensors_PZEM_data		: ARRAY[1..2] OF REAL:=2(0);

	sensors_DS18B20_id			: BYTE:=16#01;
	sensors_DS18B20_temp		: ARRAY[1..8] OF REAL:=8(0);


	get_co2_mh_z19b_1floor	: FB_GET_CO2_MH_Z19B;
(*	get_co2_mh_z19b_2floor	: FB_GET_CO2_MH_Z19B; *)
	get_co2_mh_z19b_1floor_done	: BOOL;
(*	get_co2_mh_z19b_2floor_done	: BOOL; *)
	sensor_ponics_PH_id		: BYTE:= 16#4F ;
	MBdata_sensor_ponics_PH : ARRAY [1..4] OF INT;
	Ponics_PH_temp			: REAL;

	sensor_ponics_PH_int		:INT;

	sensor_ponics_EC_id		: BYTE:= 16#51 ;
(*	sensor_ponics_EC2_id		: BYTE:= 16#50 ; *)
	sensor_ponics_EC_int		:INT;

	balkon_light_sensor_id			: BYTE:=16#5A;
	balkon_light_low				: BYTE;
	balkon_light_high				: BYTE;
	balkon_light_word				:WORD;
	balkon_light_array				: ARRAY [1..2] OF BYTE;


END_VAR
Modbus.RS485_2_cnt_error		:= CounterError;
Modbus.RS485_2_cnt_success	:= CounterSuccess;

IF (Modbus.Security_status = TRUE) THEN
	CO2_period	:= T#30m;
ELSE
	CO2_period 	:= T#2m;
END_IF



CASE state OF
	0:
		MB2.ReadRegs(Execute:= FALSE);
		state := 3;


3:
	(*	Clear2(Buffer := RxBufferCom2); *)
		MB2.ReadInputRegs(
			UnitID:=sensors_CO2_id[k], (* station address *)
			Quantity:= 1,
			MBAddr:= 3,
			cbLength:= 4,
			pMemoryAddr:= ADR(MBdata),
			Execute:= TRUE,
			Timeout:= timeoutvalue,
			Busy => busy	);
		IF NOT busy THEN
			IF (mb2.Error = FALSE ) THEN
				sensors_CO2_ppm[k]	:=	(MBdata[1]);
			END_IF
			k:=k+1;
			MB2.ReadRegs(Execute:= FALSE);
			IF (k>2 )	THEN
				k:=1;

				Modbus.Second_floor_CO2		:=	(sensors_CO2_ppm[1]);
				Modbus.First_floor_CO2		:=	(sensors_CO2_ppm[2]);
				state :=4;
			ELSE
				state :=3;
			END_IF
		END_IF



4:

		MB2.ReadInputRegs(
			UnitID:= sensors_PZEM_id,
			Quantity:= 2,
			MBAddr:= 0,
			cbLength:= 16,
			pMemoryAddr:= ADR(MBdata_pzem),
			Execute:= TRUE,
			Timeout:= timeoutvalue,
			Busy => busy,
		);
		IF NOT busy THEN
			IF (mb2.Error = FALSE ) THEN
				sensors_PZEM_data[1]:=INT_TO_REAL(MBdata_pzem[1])/100;
				sensors_PZEM_data[2]:=INT_TO_REAL(MBdata_pzem[2])/100;
				Modbus.DC_Uv:=sensors_PZEM_data[1];
				Modbus.DC_Ia:=sensors_PZEM_data[2];

			END_IF
			MB2.ReadRegs(Execute:= FALSE);
			state:=5;

		END_IF


5:

		MB2.ReadRegs(
			UnitID:= sensors_DS18B20_id,
			Quantity:= 8,
			MBAddr:= 0,
			cbLength:= 16,
			pMemoryAddr:= ADR(MBdata8),
			Execute:= TRUE,
			Timeout:= timeoutvalue,
			Busy => busy,
		);
		IF NOT busy THEN
			IF (mb2.Error = FALSE ) THEN
				sensors_DS18B20_temp[1]:=INT_TO_REAL(MBdata8[1])/10;
				sensors_DS18B20_temp[2]:=INT_TO_REAL(MBdata8[2])/10;
				sensors_DS18B20_temp[3]:=INT_TO_REAL(MBdata8[3])/10;
				sensors_DS18B20_temp[4]:=INT_TO_REAL(MBdata8[4])/10;

			END_IF
			MB2.ReadRegs(Execute:= FALSE);
			state:=17;

		END_IF

17:

		MB2.ReadRegs(
			UnitID:= balkon_light_sensor_id,
			Quantity:= 1,
			MBAddr:= 6,
			cbLength:= 2,
			pMemoryAddr:= ADR(balkon_light_array),
			Execute:= TRUE,
			Timeout:= timeoutvalue,
			Busy => busy,
		);
		IF NOT busy THEN
			IF (mb2.Error = FALSE ) THEN
				balkon_light_high:=balkon_light_array[1];
				balkon_light_low:=balkon_light_array[2];
				balkon_light_word:=(balkon_light_array[2]*256)+balkon_light_array[1];

				Modbus.Balkon_light_lux		:=	WORD_TO_UDINT(balkon_light_word);
			END_IF
			MB2.ReadRegs(Execute:= FALSE);
			state:=18;

		END_IF
18:

		MB2.ReadRegs(
			UnitID:= sensor_ponics_PH_id,
			Quantity:= 4,
			MBAddr:= 0,
			cbLength:= 8,
			pMemoryAddr:= ADR(MBdata_sensor_ponics_PH),
			Execute:= TRUE,
			Timeout:= timeoutvalue,
			Busy => busy,
		);
		IF NOT busy THEN
			IF (mb2.Error = FALSE ) THEN
				Modbus.Ponics_PH		:=	0.15+INT_TO_REAL(MBdata_sensor_ponics_PH[1])/100;
				Modbus.Ponics_tank_temp			:=	INT_TO_REAL(MBdata_sensor_ponics_PH[3])/10;

			END_IF
			MB2.ReadRegs(Execute:= FALSE);
			state:=21;

		END_IF

(*
21:

		MB2.ReadRegs(
			UnitID:= sensor_ponics_EC_id,
			Quantity:= 1,
			MBAddr:= 8,
			cbLength:= 2,
			pMemoryAddr:= ADR(sensor_ponics_EC_int),
			Execute:= TRUE,
			Timeout:= timeoutvalue,
			Busy => busy,
		);
		IF NOT busy THEN
			IF (mb2.Error = FALSE ) THEN
			Modbus.Ponics_EC	:=	-1.0 + INT_TO_REAL(sensor_ponics_EC_int)/1000;
			IF(Modbus.Ponics_EC < 0)	THEN
				Modbus.Ponics_EC	:= 0;
			END_IF

			END_IF
			MB2.ReadRegs(Execute:= FALSE);
			state:=888;

		END_IF
*)
21:

		MB2.ReadRegs(
			UnitID:= sensor_ponics_EC_id,
			Quantity:= 1,
			MBAddr:= 2,
			cbLength:= 2,
			pMemoryAddr:= ADR(sensor_ponics_EC_int),
			Execute:= TRUE,
			Timeout:= timeoutvalue,
			Busy => busy,
		);
		IF NOT busy THEN
			IF (mb2.Error = FALSE ) THEN
			Modbus.Ponics_EC	:=	 INT_TO_REAL(sensor_ponics_EC_int)/1000;
			IF(Modbus.Ponics_EC < 0)	THEN
				Modbus.Ponics_EC	:= 0;
			END_IF

			END_IF
			MB2.ReadRegs(Execute:= FALSE);
			state:=888;

		END_IF



(*	state:=105; *)
(*
105: (*открываем канал*)


	Clear(Buffer := RxBufferCom2);
	arrSend[1]:=Merc_address;
	arrSend[2]:=1; (*код доступа*)
	arrSend[3]:=1; (*Уровень доступа*)

	MEMCPY(ADR(arrSend)+3,ADR(password_1),6); (*пароль*)
	crctest:=F_CRC16(ADR(arrSend),9); (*расчет контрольной суммы*)
	MEMCPY(ADR(arrSend)+9,ADR(crctest),SIZEOF(crctest)); (*прибавление контрольной суммы к запросу*)
	SendDataCom2(pSendData:=ADR(arrSend),Length:=11,TXBuffer:=TxBufferCom2,Busy=>,Error=>);
(*	tmCheck(in:=FALSE); *)
	tmCheckM(in:=FALSE);
	tmCheckM(in:=TRUE, pt:=t#3s); 	(*запуск таймера проверки - потеря связи\обрыв кабеля*)
	state:=106;

106: (*ответ*)
	ReceiveDataCom2(pPrefix:=,LenPrefix:=,pSuffix:=,LenSuffix:=,
	pReceiveData:=ADR(arrReceive),SizeReceiveData:=4,
	Timeout:=t#2s,Reset:=,
	RXbuffer:=RxBufferCom2,
	DataReceived=>,busy=>,Error=>,RxTimeout=>,LenReceiveData=>);
	IF ReceiveDataCom2.Error <> 0 THEN
		state:=888;
	END_IF
	IF receiveDataCom2.DataReceived THEN
		state:=107;
	ELSIF tmCheckM.Q THEN
		state:=888;
	END_IF
107: (*проверка ответа*)

	IF arrReceive[1] = Merc_address THEN
		state:= 108;
	ELSE
		state:=888;
	END_IF



108:
	(*	tmCheck(in:=FALSE);	*)
		tmCheck(in:=NOT tmCheck.q,pt:=t#2s);
		get_supply_done := FALSE;
		get_supply( byte1:=16#8, byte2:=16#16, byte3:=16#11,  supply1=>Modbus.UV1,supply2=>Modbus.UV2,supply3=>Modbus.UV3, done=>get_supply_done);
		IF get_supply_done = TRUE THEN
			CounterSuccess := CounterSuccess+1;
			state:=109;
		ELSIF tmcheck.Q THEN
			CounterError := CounterError+1;
			 state:=888;
		END_IF



 (*запрос на чтение тока  на всех фазах
--------------------------------------------------------------------------------------------------------------------------------------------------------------------
*)
109:
	(*	tmCheck(in:=FALSE);	*)
		tmCheck(in:=NOT tmCheck.q,pt:=t#2s);
		get_current_done := FALSE;
		get_current(byte1:=16#8, byte2:=16#16, byte3:=16#21,  current1=>Modbus.Ia1,current2=>Modbus.Ia2,current3=>Modbus.Ia3, done=>get_current_done);
		IF get_current_done = TRUE THEN
			state:=110;
		ELSIF tmcheck.Q THEN state:=888;
		END_IF

 (*запрос на чтение мощности  на всех фазах
--------------------------------------------------------------------------------------------------------------------------------------------------------------------
*)

110:
	(*	tmCheck(in:=FALSE);	*)
		tmCheck(in:=NOT tmCheck.q,pt:=t#2s);
		get_power_done := FALSE;
		get_power(byte1:=16#8, byte2:=16#16, byte3:=16#0,  power_total=>Modbus.pw_total, power1=>Modbus.pw1, power2=>Modbus.pw2,power3=>Modbus.pw3,done=>get_power_done);
		IF get_power_done = TRUE THEN
			state:=111;
		ELSIF tmcheck.Q THEN state:=888;
		END_IF

 (*запрос на чтение энергии T1
--------------------------------------------------------------------------------------------------------------------------------------------------------------------
*)
111:
	(*	tmCheck(in:=FALSE);	*)
		tmCheck(in:=NOT tmCheck.q,pt:=t#2s);
		get_energy_E_T1_done := FALSE;
		get_energy_E_T1(byte1:=5, byte2:=16#0, byte3:=1,  energy=>Modbus.E_T1, done=>get_energy_E_T1_done);
		IF get_energy_E_T1_done = TRUE THEN
			state:=112;
		ELSIF tmcheck.Q THEN state:=888;
		END_IF
 (*запрос на чтение энергии T2
--------------------------------------------------------------------------------------------------------------------------------------------------------------------
*)

112:
	(*	tmCheck(in:=FALSE);	*)
		tmCheck(in:=NOT tmCheck.q,pt:=t#2s);
		get_energy_E_T2_done := FALSE;
		get_energy_E_T2(byte1:=5, byte2:=16#0, byte3:=2,  energy=>Modbus.E_T2, done=>get_energy_E_T2_done);
		IF get_energy_E_T2_done = TRUE THEN
			state:=113;
		ELSIF tmcheck.Q THEN state:=888;
		END_IF

113:
		Timer_day(IN:=NOT Timer_dayQ , PT:=T#30m , Q=>Timer_dayQ , ET=> );
			IF timer_day.q THEN
				state:=114;
			ELSE
				state:=888;
			END_IF

114:
	(*	tmCheck(in:=FALSE);	*)
		tmCheckE(in:=NOT tmCheckE.q,pt:=t#2s, Q=>tmCheckEQ , ET=>);
		get_energy_MT_done := FALSE;

	(*	IF (tmCheckEQ) THEN *)
			get_energy_MT(byte1:=5, byte2:=INT_TO_BYTE(48+m), byte3:=INT_TO_BYTE(t),   energy=>energyMT[m,t],done=>get_energy_MT_done);
(*		END_IF *)

		IF get_energy_MT_done = TRUE THEN
			t:=t+1;
			IF (t>2 AND m<13) THEN
				t:=1;
				m:=m+1;
				state:=114;
			END_IF

					IF ( m=13) THEN
						t:=1;
						m:=1;
						Modbus.M1T1:=energyMT[1,1];
						Modbus.M1T2:=energyMT[1,2];
						Modbus.M2T1:=energyMT[2,1];
						Modbus.M2T2:=energyMT[2,2];
						Modbus.M3T1:=energyMT[3,1];
						Modbus.M3T2:=energyMT[3,2];
						Modbus.M4T1:=energyMT[4,1];
						Modbus.M4T2:=energyMT[4,2];
						Modbus.M5T1:=energyMT[5,1];
						Modbus.M5T2:=energyMT[5,2];
						Modbus.M6T1:=energyMT[6,1];
						Modbus.M6T2:=energyMT[6,2];
						Modbus.M7T1:=energyMT[7,1];
						Modbus.M7T2:=energyMT[7,2];
						Modbus.M8T1:=energyMT[8,1];
						Modbus.M8T2:=energyMT[8,2];
						Modbus.M9T1:=energyMT[9,1];
						Modbus.M9T2:=energyMT[9,2];
						Modbus.M10T1:=energyMT[10,1];
						Modbus.M10T2:=energyMT[10,2];
						Modbus.M11T1:=energyMT[11,1];
						Modbus.M11T2:=energyMT[11,2];
						Modbus.M12T1:=energyMT[12,1];
						Modbus.M12T2:=energyMT[12,2];
						state:=888;
					END_IF
		ELSIF tmcheckE.Q THEN state:=114;
		END_IF


*)


888:
		TimerRS485_2(IN:=NOT TimerRS485_2Q , PT:=tTimerValue , Q=>TimerRS485_2Q , ET=> );
		IF TimerRS485_2.q THEN
			state:=0;
		END_IF

END_CASE

FtrigBusy(CLK:=mb2.BUSY );
IF FtrigBusy.Q THEN
	IF mb2.Error THEN
		LastModbusError := mb2.ErrorDiagnostics;
		LastErrorstate := state;
		CounterError := CounterError + 1;
	ELSE
		CounterSuccess := CounterSuccess + 1;
	END_IF
END_IF

SerialLinecontrolCom2(
	mode:=SerialLinemode_kl6_5b_standard,
	pComIn:=ADR(RS485read_2.MB2.InData),
	pComOut:=ADR(RS485read_2.MB2.OutData),
	SizeComIn:=SIZEOF(RS485read_2.MB2.OutData),
	TxBuffer:=TxBufferCom2,
	RxBuffer:=RxBufferCom2,
	Error=>,
	errorid=>);
END_PROGRAM

(* POU FB_GET_CO2_MH_Z19B, ST *)
FUNCTION_BLOCK FB_GET_CO2_MH_Z19B
VAR_INPUT

END_VAR

VAR_OUTPUT
	co2				: REAL;
	done			: BOOL;
END_VAR

VAR
	SendBuffer		: ARRAY[0..8] OF BYTE;
	ReceiveBuffer	: ARRAY[0..13] OF BYTE;
	Clear			: ClearComBuffer;
	state			: INT:= 0;
	tmcheck			: TON;
	w_CO2		:	WORD;
END_VAR
tmcheck();

CASE state OF

0:
	done:=FALSE;
	Clear(Buffer := RxBufferCom1);
	SendBuffer[0] := 16#FF;
	SendBuffer[1] := 16#01; (* Address *)
	SendBuffer[2] := 16#86;
	SendBuffer[3] := 16#00;
	SendBuffer[4] := 16#00;
	SendBuffer[5] := 16#00;
	SendBuffer[6] := 16#00;
	SendBuffer[7] := 16#00;	(* Checksum *)
	SendBuffer[8] := 16#79;	(* Checksum *)

	SendDataCom1(pSendData:=ADR(SendBuffer),length:=9,TXbuffer:=TXBufferCom1,Busy=>,Error=>);

	tmCheck(in:=FALSE);
	tmCheck(in:=TRUE,pt:=t#2s);
	state:=1;

1: (*ответ*)

	ReceiveDataCom1(pPrefix:=,LenPrefix:=,pSuffix:=,LenSuffix:=,pReceiveData:=ADR(ReceiveBuffer),SizeReceiveData:=9,TImeOut:=t#1s,Reset:=,RXbuffer:=RxBufferCom1,DataReceived=>,busy=>,RxTimeout=>,LenReceiveData=>);

	IF ReceiveDataCom1.Error <> 0 THEN
		state:=9;
	END_IF

	IF ReceiveDataCom1.DataReceived THEN
		state:=2;
	ELSIF tmcheck.Q THEN
		 state:=9;
	END_IF;



2:(*расшифровка*)
	IF (ReceiveBuffer [0] = 16#FF AND ReceiveBuffer [1] = 16#86 ) THEN
		Sensor_CO2_high := ReceiveBuffer [2];
		Sensor_CO2_low := ReceiveBuffer [3];
		MEMCPY(ADR(w_CO2),ADR(ReceiveBuffer[3]),1);
		MEMCPY(ADR(w_CO2)+1,ADR(ReceiveBuffer[2]),1);
		IF (WORD_TO_REAL(w_CO2)<>0 AND WORD_TO_REAL(w_CO2)<5001) THEN
			co2 := WORD_TO_REAL(w_CO2);
			state:=10;
		ELSE
			state:=9;
		END_IF
	ELSE
		state:=9;
	END_IF

9:
	co2:=0;
	done := TRUE;
	state:=0;
10:
	done := TRUE;
	state:=0;

END_CASE;
END_FUNCTION_BLOCK

(* POU RS485read_3, ST *)
PROGRAM RS485read_3
VAR

	tTimerValue			: TIME	:=	t#30s; (* Период опроса RS485*)

(*	password_1				: ARRAY [1..6] OF BYTE:=6(1); (* пароль к меркуриям, по умолчанию 6 единиц*)
	crctest					: WORD;
	arrReceive				: ARRAY[1..22] OF BYTE;
	arrSend					: ARRAY[1..22] OF BYTE;
*)
	MBdata					 : ARRAY [1..2] OF INT;
	FtrigBusy				: F_TRIG;
	timeoutvalue				: TIME := T#1000ms;		(* timeout while waiting for an answer of the modbus slave *)
	state					: INT;
	busy					: BOOL;
	LastErrorstate				: INT;
	LastModbusError			: ST_ModbusErrorDiagnostics;
	CounterError				: DINT;
	CounterSuccess			: DINT;
	teplica_DS18B20_id			: BYTE:=16#44;
	teplica_DS18B20_temp		: ARRAY[1..8] OF REAL:=8(0);
	MBdata8					 : ARRAY [1..8] OF UINT;
(*	teplica_ADM4188_id			: BYTE:=16#45; *)
	teplica_light_sensor_id			: BYTE:=16#3C;
	teplica_light_low				: WORD;
	teplica_light_high				: WORD;
	teplica_light_dword				:DWORD;
	teplica_light_array				: ARRAY [1..2] OF WORD;
	sensors_SHT30_v3_id			:  BYTE:= 16#32 ;
	sensors_SHT30_v3_hum		:  REAL;
	sensors_SHT30_v3_temp		:  REAL;
	sensor_teplica_PH_id		: BYTE:= 16#78 ;
	sensor_teplica_EC_id			: BYTE:= 16#C8 ;
	MBdata_sensor_teplica_EC		 : ARRAY [1..4] OF INT;
	password_1				: ARRAY [1..6] OF BYTE:=6(1); (* пароль к меркуриям, по умолчанию 6 единиц*)
	crctest					: WORD;
	get_energy_E_T1			: FB_GET_ENERGY;
	get_energy_E_T2			: FB_GET_ENERGY;
	get_energy_MT			: FB_GET_ENERGY;
	get_supply				: FB_GET_SUPPLY;
	get_current				: FB_GET_CURRENT;
	get_power				: FB_GET_POWER;
	energyMT					: ARRAY[1..12,1..2] OF REAL;
	get_current_done			: BOOL;
	get_power_done			: BOOL;
	get_energy_E_T1_done	: BOOL;
	get_energy_E_T2_done	: BOOL;
	get_energy_MT_done		: BOOL;

	get_supply_done			: BOOL;
	arrReceive				: ARRAY[1..5] OF BYTE;
	arrSend					: ARRAY[1..5] OF BYTE;
	t,m						: INT:=1;
	MBdata_sensor_ponics_PH : ARRAY [1..4] OF INT;
	Teplica_ph_sensor_temp	: REAL;

END_VAR
Modbus.RS485_3_cnt_error		:= CounterError;
Modbus.RS485_3_cnt_success	:= CounterSuccess;





CASE state OF
0:
	MB3.ReadRegs(Execute:= FALSE);
	state :=888;




15:

		MB3.ReadRegs(
			UnitID:= teplica_DS18B20_id,
			Quantity:= 8,
			MBAddr:= 0,
			cbLength:= 16,
			pMemoryAddr:= ADR(MBdata8),
			Execute:= TRUE,
			Timeout:=  T#2000ms,
			Busy => busy,
		);
		IF NOT busy THEN
			IF (mb3.Error = FALSE ) THEN
				IF (MBdata8[1] < 10000)
					THEN	teplica_DS18B20_temp[1]:=UINT_TO_REAL(MBdata8[1])/10;
				ELSE
					teplica_DS18B20_temp[1]:=-1*UINT_TO_REAL(MBdata8[1]-10000)/10;
				END_IF

				IF (MBdata8[2] < 10000)
					THEN	teplica_DS18B20_temp[2]:=UINT_TO_REAL(MBdata8[2])/10;
				ELSE
					teplica_DS18B20_temp[2]:=-1*UINT_TO_REAL(MBdata8[2]-10000)/10;
				END_IF


				IF (MBdata8[3] < 10000)
					THEN	teplica_DS18B20_temp[3]:=UINT_TO_REAL(MBdata8[3])/10;
				ELSE
					teplica_DS18B20_temp[3]:=-1*UINT_TO_REAL(MBdata8[3]-10000)/10;
				END_IF

				IF (MBdata8[4] < 10000)
					THEN	teplica_DS18B20_temp[4]:=UINT_TO_REAL(MBdata8[4])/10;
				ELSE
					teplica_DS18B20_temp[4]:=-1*UINT_TO_REAL(MBdata8[4]-10000)/10;
				END_IF

				IF  (teplica_DS18B20_temp[1] <>0 AND teplica_DS18B20_temp[1] <>85)	THEN
					Modbus.Teplica_temp_air			:=	teplica_DS18B20_temp[1];
				END_IF

				IF  (teplica_DS18B20_temp[2] <>0 AND teplica_DS18B20_temp[2] <>85)	THEN
					Modbus.Teplica_temp_ground		:=	teplica_DS18B20_temp[2];
				END_IF

				IF  (teplica_DS18B20_temp[3] <>0 AND teplica_DS18B20_temp[3] <>85)	THEN
					Modbus.Teplica_temp_pipe_heat 	:=	teplica_DS18B20_temp[3];
				END_IF

				IF  (teplica_DS18B20_temp[4] <>0 AND teplica_DS18B20_temp[4] <>85)	THEN
					Modbus.Teplica_temp_water_tank 	:=	teplica_DS18B20_temp[4];
				END_IF


			END_IF
			MB3.ReadRegs(Execute:= FALSE);
			state:=16;

		END_IF


16:

		MB3.ReadRegs(
			UnitID:= teplica_light_sensor_id,
			Quantity:= 2,
			MBAddr:= 2,
			cbLength:= 4,
			pMemoryAddr:= ADR(teplica_light_array),
			Execute:= TRUE,
			Timeout:= timeoutvalue,
			Busy => busy,
		);
		IF NOT busy THEN
			IF (mb3.Error = FALSE ) THEN
				teplica_light_high:=teplica_light_array[1];
				teplica_light_low:=teplica_light_array[2];
				teplica_light_dword:=(teplica_light_array[1]*65535)+teplica_light_array[2];

				Modbus.Teplica_light_lux		:=	DWORD_TO_REAL(teplica_light_dword);


			END_IF
			MB3.ReadRegs(Execute:= FALSE);
			state:=18;

		END_IF





18:
		MB3.ReadRegs(
			UnitID:= sensors_SHT30_v3_id,
			Quantity:= 2,
			MBAddr:= 512,
			cbLength:= 6,
			pMemoryAddr:= ADR(MBdata),
			Execute:= TRUE,
			Timeout:= timeoutvalue,
			Busy => busy,
		);
		IF NOT busy THEN
			IF (mb3.Error = FALSE ) THEN
				sensors_SHT30_v3_temp:=INT_TO_REAL(MBdata[1])/10;
				sensors_SHT30_v3_hum:=INT_TO_REAL(MBdata[2])/10;

				Internal.Teplica_temp_SHT30		:=	sensors_SHT30_v3_temp;
				Internal.Teplica_hum_SHT30		:=	sensors_SHT30_v3_hum;
				Modbus.Teplica_temp_SHT30		:=	sensors_SHT30_v3_temp;
				Modbus.Teplica_hum_SHT30		:=	sensors_SHT30_v3_hum;
			END_IF
			MB3.ReadRegs(Execute:= FALSE);
			state :=19;
		END_IF

19:

		MB3.ReadRegs(
			UnitID:= sensor_teplica_PH_id,
			(*Quantity:= 1,
			MBAddr:= 0,
			cbLength:= 2,
			pMemoryAddr:= ADR(sensor_teplica_PH_int),*)
			Quantity:= 4,
			MBAddr:= 0,
			cbLength:= 8,
			pMemoryAddr:= ADR(MBdata_sensor_ponics_PH),
			Execute:= TRUE,
			Timeout:= timeoutvalue,
			Busy => busy,
		);
		IF NOT busy THEN
			IF (mb3.Error = FALSE ) THEN

(*				Modbus.Teplica_sensor_soil_PH		:=	INT_TO_REAL(sensor_teplica_PH_int)/100;	*)
				Modbus.Teplica_sensor_soil_PH	:=	INT_TO_REAL(MBdata_sensor_ponics_PH[1])/100;
				Teplica_ph_sensor_temp			:=	INT_TO_REAL(MBdata_sensor_ponics_PH[3])/10;

			END_IF
			MB3.ReadRegs(Execute:= FALSE);
			state:=20;

		END_IF

20:

		MB3.ReadRegs(
			UnitID:= sensor_teplica_EC_id,
			Quantity:= 4,
			MBAddr:= 0,
			cbLength:= 8,
			pMemoryAddr:= ADR(MBdata_sensor_teplica_EC),
			Execute:= TRUE,
			Timeout:= timeoutvalue,
			Busy => busy,
		);
		IF NOT busy THEN
			IF (mb3.Error = FALSE ) THEN
			Modbus.Teplica_sensor_soil_Hum	:=	INT_TO_REAL(MBdata_sensor_teplica_EC[1])/10;
			Modbus.Teplica_sensor_soil_Temp	:=	INT_TO_REAL(MBdata_sensor_teplica_EC[2])/10;
			Modbus.Teplica_sensor_soil_EC	:=	INT_TO_REAL(MBdata_sensor_teplica_EC[3]);
			Modbus.Teplica_sensor_soil_PH2	:=	INT_TO_REAL(MBdata_sensor_teplica_EC[4])/10;

			END_IF
			MB3.ReadRegs(Execute:= FALSE);
			state:=105;

		END_IF



(*	state:=105; *)

105: (*открываем канал*)


	Clear(Buffer := RxBufferCom3);
	arrSend[1]:=Merc_address;
	arrSend[2]:=1; (*код доступа*)
	arrSend[3]:=1; (*Уровень доступа*)

	MEMCPY(ADR(arrSend)+3,ADR(password_1),6); (*пароль*)
	crctest:=F_CRC16(ADR(arrSend),9); (*расчет контрольной суммы*)
	MEMCPY(ADR(arrSend)+9,ADR(crctest),SIZEOF(crctest)); (*прибавление контрольной суммы к запросу*)
	SendDataCom3(pSendData:=ADR(arrSend),Length:=11,TXBuffer:=TxBufferCom3,Busy=>,Error=>);
(*	tmCheck(in:=FALSE); *)
	tmCheckM(in:=FALSE);
	tmCheckM(in:=TRUE, pt:=t#3s); 	(*запуск таймера проверки - потеря связи\обрыв кабеля*)
	state:=106;

106: (*ответ*)
	ReceiveDataCom3(pPrefix:=,LenPrefix:=,pSuffix:=,LenSuffix:=,
	pReceiveData:=ADR(arrReceive),SizeReceiveData:=4,
	Timeout:=t#2s,Reset:=,
	RXbuffer:=RxBufferCom3,
	DataReceived=>,busy=>,Error=>,RxTimeout=>,LenReceiveData=>);
	IF ReceiveDataCom3.Error <> 0 THEN
		state:=888;
	END_IF
	IF receiveDataCom3.DataReceived THEN
		state:=107;
	ELSIF tmCheckM.Q THEN
		state:=888;
	END_IF
107: (*проверка ответа*)

	IF arrReceive[1] = Merc_address THEN
		state:= 108;
	ELSE
		state:=888;
	END_IF



108:
	(*	tmCheck(in:=FALSE);	*)
		tmCheck(in:=NOT tmCheck.q,pt:=t#2s);
		get_supply_done := FALSE;
		get_supply( byte1:=16#8, byte2:=16#16, byte3:=16#11,  supply1=>Modbus.UV1,supply2=>Modbus.UV2,supply3=>Modbus.UV3, done=>get_supply_done);
		IF get_supply_done = TRUE THEN
			CounterSuccess := CounterSuccess+1;
			state:=109;
		ELSIF tmcheck.Q THEN
			CounterError := CounterError+1;
			 state:=888;
		END_IF



 (*запрос на чтение тока  на всех фазах
--------------------------------------------------------------------------------------------------------------------------------------------------------------------
*)
109:
	(*	tmCheck(in:=FALSE);	*)
		tmCheck(in:=NOT tmCheck.q,pt:=t#2s);
		get_current_done := FALSE;
		get_current(byte1:=16#8, byte2:=16#16, byte3:=16#21,  current1=>Modbus.Ia1,current2=>Modbus.Ia2,current3=>Modbus.Ia3, done=>get_current_done);
		IF get_current_done = TRUE THEN
			state:=110;
		ELSIF tmcheck.Q THEN state:=888;
		END_IF

 (*запрос на чтение мощности  на всех фазах
--------------------------------------------------------------------------------------------------------------------------------------------------------------------
*)

110:
	(*	tmCheck(in:=FALSE);	*)
		tmCheck(in:=NOT tmCheck.q,pt:=t#2s);
		get_power_done := FALSE;
		get_power(byte1:=16#8, byte2:=16#16, byte3:=16#0,  power_total=>Modbus.pw_total, power1=>Modbus.pw1, power2=>Modbus.pw2,power3=>Modbus.pw3,done=>get_power_done);
		IF get_power_done = TRUE THEN
			state:=111;
		ELSIF tmcheck.Q THEN state:=888;
		END_IF

 (*запрос на чтение энергии T1
--------------------------------------------------------------------------------------------------------------------------------------------------------------------
*)
111:
	(*	tmCheck(in:=FALSE);	*)
		tmCheck(in:=NOT tmCheck.q,pt:=t#2s);
		get_energy_E_T1_done := FALSE;
		get_energy_E_T1(byte1:=5, byte2:=16#0, byte3:=1,  energy=>Modbus.E_T1, done=>get_energy_E_T1_done);
		IF get_energy_E_T1_done = TRUE THEN
			state:=112;
		ELSIF tmcheck.Q THEN state:=888;
		END_IF
 (*запрос на чтение энергии T2
--------------------------------------------------------------------------------------------------------------------------------------------------------------------
*)

112:
	(*	tmCheck(in:=FALSE);	*)
		tmCheck(in:=NOT tmCheck.q,pt:=t#2s);
		get_energy_E_T2_done := FALSE;
		get_energy_E_T2(byte1:=5, byte2:=16#0, byte3:=2,  energy=>Modbus.E_T2, done=>get_energy_E_T2_done);
		IF get_energy_E_T2_done = TRUE THEN
			state:=888;
		ELSIF tmcheck.Q THEN state:=888;
		END_IF

113:
		Timer_day(IN:=NOT Timer_dayQ , PT:=T#30m , Q=>Timer_dayQ , ET=> );
			IF timer_day.q THEN
				state:=114;
			ELSE
				state:=888;
			END_IF

114:
	(*	tmCheck(in:=FALSE);	*)
		tmCheckE(in:=NOT tmCheckE.q,pt:=t#2s, Q=>tmCheckEQ , ET=>);
		get_energy_MT_done := FALSE;

	(*	IF (tmCheckEQ) THEN *)
			get_energy_MT(byte1:=5, byte2:=INT_TO_BYTE(48+m), byte3:=INT_TO_BYTE(t),   energy=>energyMT[m,t],done=>get_energy_MT_done);
(*		END_IF *)

		IF get_energy_MT_done = TRUE THEN
			t:=t+1;
			IF (t>2 AND m<13) THEN
				t:=1;
				m:=m+1;
				state:=114;
			END_IF

					IF ( m=13) THEN
						t:=1;
						m:=1;
						Modbus.M1T1:=energyMT[1,1];
						Modbus.M1T2:=energyMT[1,2];
						Modbus.M2T1:=energyMT[2,1];
						Modbus.M2T2:=energyMT[2,2];
						Modbus.M3T1:=energyMT[3,1];
						Modbus.M3T2:=energyMT[3,2];
						Modbus.M4T1:=energyMT[4,1];
						Modbus.M4T2:=energyMT[4,2];
						Modbus.M5T1:=energyMT[5,1];
						Modbus.M5T2:=energyMT[5,2];
						Modbus.M6T1:=energyMT[6,1];
						Modbus.M6T2:=energyMT[6,2];
						Modbus.M7T1:=energyMT[7,1];
						Modbus.M7T2:=energyMT[7,2];
						Modbus.M8T1:=energyMT[8,1];
						Modbus.M8T2:=energyMT[8,2];
						Modbus.M9T1:=energyMT[9,1];
						Modbus.M9T2:=energyMT[9,2];
						Modbus.M10T1:=energyMT[10,1];
						Modbus.M10T2:=energyMT[10,2];
						Modbus.M11T1:=energyMT[11,1];
						Modbus.M11T2:=energyMT[11,2];
						Modbus.M12T1:=energyMT[12,1];
						Modbus.M12T2:=energyMT[12,2];
						state:=888;
					END_IF
		ELSIF tmcheckE.Q THEN state:=114;
		END_IF






888:
		TimerRS485_3(IN:=NOT TimerRS485_3Q , PT:=tTimerValue , Q=>TimerRS485_3Q , ET=> );
		IF TimerRS485_3.q THEN
			state:=0;
		END_IF


END_CASE

FtrigBusy(CLK:=mb3.BUSY );
IF FtrigBusy.Q THEN
	IF mb3.Error THEN
		LastModbusError := mb3.ErrorDiagnostics;
		LastErrorstate := state;
		CounterError := CounterError + 1;
	ELSE
		CounterSuccess := CounterSuccess + 1;
	END_IF
END_IF



SerialLinecontrolCom3(
	mode:=SerialLinemode_kl6_22b_standard,
	pComIn:=ADR(RS485read_3.MB3.InData),
	pComOut:=ADR(RS485read_3.MB3.OutData),
	SizeComIn:=SIZEOF(RS485read_3.MB3.OutData),
	TxBuffer:=TxBufferCom3,
	RxBuffer:=RxBufferCom3,
	Error=>,
	errorid=>);
END_PROGRAM

(* POU RS485read_3_old, ST *)
PROGRAM RS485read_3_old
VAR
(*	Period_vent_switch	: INT:=180; *)

	tTimerValue			: TIME	:=	t#10s; (* Период опроса RS485*)

(*	password_1				: ARRAY [1..6] OF BYTE:=6(1); (* пароль к меркуриям, по умолчанию 6 единиц*)
	crctest					: WORD;
	arrReceive				: ARRAY[1..22] OF BYTE;
	arrSend					: ARRAY[1..22] OF BYTE;
*)
	MBdata					 : ARRAY [1..2] OF INT;
	FtrigBusy				: F_TRIG;
	timeoutvalue				: TIME := T#1000ms;		(* timeout while waiting for an answer of the modbus slave *)
	state					: INT;
	busy					: BOOL;
	LastErrorstate				: INT;
	LastModbusError			: ST_ModbusErrorDiagnostics;
	CounterError				: DINT;
	CounterSuccess			: DINT;
	CounterError_M			: DINT;
	CounterSuccess_M		: DINT;

(*	i,k,l,m,t					: INT:=1; *)





	teplica_DS18B20_id			: BYTE:=16#44;
	teplica_DS18B20_temp		: ARRAY[1..8] OF REAL:=8(0);
	MBdata8					 : ARRAY [1..8] OF UINT;

(*	Modbus_DO					: INT:=1; *)
	teplica_ADM4188_id			: BYTE:=16#45;
(*	teplica_ADM4188_DI_1			:  INT;
	teplica_ADM4188_DO_1		:  INT;
	teplica_ADM4188_DO_1_ACK	:  INT; *)

	teplica_light_sensor_id			: BYTE:=16#3C;
	teplica_light_low				: WORD;
	teplica_light_high				: WORD;
	teplica_light_dword				:DWORD;
	teplica_light_array				: ARRAY [1..2] OF WORD;


	balkon_light_sensor_id			: BYTE:=16#5A;
	balkon_light_low				: BYTE;
	balkon_light_high				: BYTE;
	balkon_light_word				:WORD;
	balkon_light_array				: ARRAY [1..2] OF BYTE;






	MBdataDI		 			 : ARRAY [1..8] OF UINT;
	MBdataDO_byte					: INT;
	MBdataDO_byte_old				: INT;


(*	teplica_ADM4188_DO_ACK		:  INT;
	teplica_ADM4188_DI_ACK		: INT; *)
(*	teplica_ADM4188_DO_1		:  INT; *)

	zero						: INT:=0;



(*	TRIG_start_reset			:	R_TRIG; *)

	Teplica_DI1_cnt			:	UINT;
	Teplica_DI2_cnt			:	UINT;
	Teplica_DI3_cnt			:	UINT;
	Teplica_DI1_cnt_mem		:	UINT;
	Teplica_DI2_cnt_mem		:	UINT;
	Teplica_DI3_cnt_mem		:	UINT;

	check0					: INT:=0;
	check1					: INT:=0;
	check2					: INT:=0;
	check3					: INT:=0;

	sensors_SHT30_v3_id			:  BYTE:= 16#32 ;
	sensors_SHT30_v3_hum		:  REAL;
	sensors_SHT30_v3_temp		:  REAL;

	sensor_teplica_PH_id			: BYTE:= 16#78 ;
	sensor_teplica_PH_int		:INT;

	sensor_teplica_EC_id			: BYTE:= 16#C8 ;
	MBdata_sensor_teplica_EC		 : ARRAY [1..4] OF INT;

	cnt_clear_di_1			: BOOL;
	cnt_clear_di_2			: BOOL;
	cnt_clear_di_3			: BOOL;
	cnt_overload_1			:INT;
	cnt_overload_2			:INT;
	cnt_overload_3			:INT;

END_VAR
Modbus.RS485_3_cnt_error		:= CounterError;
Modbus.RS485_3_cnt_success	:= CounterSuccess;


MBdataDO_byte.0			:=	Modbus.Teplica_DO1_vent;
MBdataDO_byte.1			:=	Modbus.Teplica_DO2_heat;
MBdataDO_byte.2			:=	Modbus.Teplica_DO3_light;
MBdataDO_byte.3			:=	Modbus.Teplica_DO4_pomp_poliv;
MBdataDO_byte.4			:=	Modbus.Teplica_DO5_pomp_fertA;
MBdataDO_byte.5			:=	Modbus.Teplica_DO6_pomp_fertB;
MBdataDO_byte.6			:=	Modbus.Teplica_DO7;
MBdataDO_byte.7			:=	Modbus.Teplica_DO8;



CASE state OF
0:
MB3.ReadRegs(Execute:= FALSE);

IF (Modbus.Teplica_poliv_status_PLC =1 )   THEN
	state := 1;
	check0:=check0+1;
ELSE
	state :=9;
END_IF




1:
(*Обнуление счётчиков полива и фертигации при старте полива*)

	Modbus.Teplica_poliv_message_PLC	:=	1;
	Modbus.Teplica_poliv_status_PLC 		:=	4;
	check1:=check1+1;
	cnt_clear_di_1	:= FALSE;
	MB3.WriteSingleRegister(
					UnitID:= teplica_ADM4188_id, (* station address *)
					Quantity:= 1,
					MBAddr:= 0,
					cbLength:= 2,
					pMemoryAddr:= ADR(zero),
					Execute:= TRUE,
					Timeout:= T#2000ms,
					Busy => busy,
					);
		IF NOT busy THEN
			IF (mb3.Error = FALSE ) THEN
					Modbus.Teplica_poliv_message_PLC	:=	2;
					Cnt_Teplica_poliv_message_PLC_M3	:=	0;
					cnt_clear_di_1	:=	TRUE;


			END_IF
			IF (mb3.Error = TRUE ) THEN
					Modbus.Teplica_DI1_poliv				:=	0;
					cnt_clear_di_1	:=	FALSE;
					Cnt_Teplica_poliv_message_PLC_M3	 :=	Cnt_Teplica_poliv_message_PLC_M3+1;
					Cnt_Teplica_poliv_status_PLC_N3		:=	Cnt_Teplica_poliv_status_PLC_N3+1;
					IF (Cnt_Teplica_poliv_message_PLC_M3 >2) THEN
						Modbus.Teplica_poliv_status_PLC		:=	3;
						Modbus.Teplica_poliv_message_PLC	:=	3;
					END_IF

			END_IF


			MB3.ReadRegs(Execute:= FALSE);
			state:=2;
		END_IF

2:
	check2:=check2+1;
	cnt_clear_di_2	:=	FALSE;

	MB3.WriteSingleRegister(
					UnitID:= teplica_ADM4188_id, (* station address *)
					Quantity:= 1,
					MBAddr:= 1,
					cbLength:= 2,
					pMemoryAddr:= ADR(zero),
					Execute:= TRUE,
					Timeout:= T#2000ms,
					Busy => busy,
					);
		IF NOT busy THEN
			IF (mb3.Error = FALSE ) THEN
					Modbus.Teplica_poliv_message_PLC	:=	4;
					Cnt_Teplica_poliv_message_PLC_M5	 :=	0;
					Modbus.Teplica_DI2_fertA				:=	0;
					cnt_clear_di_2	:=	TRUE;

			END_IF
			IF (mb3.Error = TRUE ) THEN
					Cnt_Teplica_poliv_message_PLC_M5	 :=	Cnt_Teplica_poliv_message_PLC_M5+1;
					cnt_clear_di_2	:=	FALSE;
					IF (Cnt_Teplica_poliv_message_PLC_M5 >2) THEN
						Modbus.Teplica_poliv_status_PLC		:=	3;
						Modbus.Teplica_poliv_message_PLC	:=	5;
					END_IF

			END_IF
			MB3.ReadRegs(Execute:= FALSE);
			state:=3;
		END_IF

3:
		check3:=check3+1;
		cnt_clear_di_3	:=	FALSE;
		MB3.WriteSingleRegister(
					UnitID:= teplica_ADM4188_id, (* station address *)
					Quantity:= 1,
					MBAddr:= 2,
					cbLength:= 2,
					pMemoryAddr:= ADR(zero),
					Execute:= TRUE,
					Timeout:= T#2000ms,
					Busy => busy,
					);
		IF NOT busy THEN
			IF (mb3.Error = FALSE ) THEN
					Modbus.Teplica_poliv_status_PLC	:=	2;
					Modbus.Teplica_poliv_message_PLC	:=	6;
					Cnt_Teplica_poliv_message_PLC_M7	 :=	0;
					Modbus.Teplica_DI3_fertB				:=	0;
					cnt_clear_di_3	:=	TRUE;
					IF (cnt_clear_di_1 = TRUE AND cnt_clear_di_2 = TRUE AND cnt_clear_di_3 = TRUE ) THEN
						Teplica_DI1_cnt_mem		:=0;
						Teplica_DI2_cnt_mem		:=0;
						Teplica_DI3_cnt_mem		:=0;
						cnt_overload_1			:=0;
						cnt_overload_2			:=0;
						cnt_overload_3			:=0;
						Cnt_cleared	:=	TRUE;
					END_IF

			END_IF
			IF (mb3.Error = TRUE ) THEN
					Cnt_Teplica_poliv_message_PLC_M7	 :=	Cnt_Teplica_poliv_message_PLC_M7+1;
					cnt_clear_di_3	:=	FALSE;
					IF (Cnt_Teplica_poliv_message_PLC_M7 >2) THEN
						Modbus.Teplica_poliv_status_PLC		:=	3;
						Modbus.Teplica_poliv_message_PLC	:=	7;
					END_IF

			END_IF
			MB3.ReadRegs(Execute:= FALSE);
			state:=9;
		END_IF

(*Запись DO значений*)


(*считывание DI значений *)
9:
	MB3.ReadRegs(
					UnitID:= teplica_ADM4188_id, (* station address *)
					Quantity:= 8,
					MBAddr:= 0,
					cbLength:= 16,
					pMemoryAddr:= ADR(MBdataDI),
					Execute:= TRUE,
					Timeout:= T#2000ms,
					Busy => busy,
					);
		IF NOT busy THEN
			IF (mb3.Error = FALSE ) THEN
					Modbus.Teplica_poliv_message_PLC	:=	10;
					Teplica_DI1_cnt	:=MBdataDI[1];
					Teplica_DI2_cnt	:=MBdataDI[2];
					Teplica_DI3_cnt	:=MBdataDI[3];

			IF (Cnt_cleared = TRUE) THEN
				IF ( Teplica_DI1_cnt_mem > Teplica_DI1_cnt AND Teplica_DI1_cnt_mem > 50000)  THEN
					cnt_overload_1	:=	cnt_overload_1+1;
					Modbus.Teplica_DI1_poliv	:= Modbus.Teplica_DI1_poliv + (65535-Teplica_DI1_cnt_mem);
				END_IF
				Modbus.Teplica_DI1_poliv	:= cnt_overload_1*65535+Teplica_DI1_cnt;


				IF ( Teplica_DI2_cnt_mem > Teplica_DI2_cnt AND Teplica_DI2_cnt_mem > 50000)   THEN
					cnt_overload_2	:=	cnt_overload_2+1;
					Modbus.Teplica_DI2_fertA	:= Modbus.Teplica_DI2_fertA + (65535-Teplica_DI2_cnt_mem);
				END_IF
				Modbus.Teplica_DI2_fertA	:= cnt_overload_2*65535+Teplica_DI2_cnt;


				IF ( Teplica_DI3_cnt_mem > Teplica_DI3_cnt AND Teplica_DI3_cnt_mem > 50000)  THEN
					cnt_overload_3	:=	cnt_overload_3+1;
					Modbus.Teplica_DI3_fertB	:= Modbus.Teplica_DI3_fertB + (65535-Teplica_DI3_cnt_mem);
				END_IF
				Modbus.Teplica_DI3_fertB	:= cnt_overload_3*65535+Teplica_DI3_cnt;

				Teplica_DI1_cnt_mem		:=Teplica_DI1_cnt;
				Teplica_DI2_cnt_mem		:=Teplica_DI2_cnt;
				Teplica_DI3_cnt_mem		:=Teplica_DI3_cnt;

				IF (Modbus.Teplica_DO5_pomp_fertA =  TRUE OR FertA_init_stop = TRUE) THEN
					Modbus.Cnt_water_fertA	:=	Modbus.Teplica_DI1_poliv -Cnt_water_fertA_start;
				END_IF

				IF (Modbus.Teplica_DO6_pomp_fertB =  TRUE OR FertB_init_stop = TRUE) THEN
					Modbus.Cnt_water_fertB	:=	Modbus.Teplica_DI1_poliv -Cnt_water_fertB_start;
				END_IF

			END_IF

				Cnt_Teplica_poliv_message_PLC_M11	 :=	0;

			END_IF

			IF (mb3.Error = TRUE ) THEN

					Cnt_Teplica_poliv_message_PLC_M11	 :=	Cnt_Teplica_poliv_message_PLC_M11+1;
					IF (Cnt_Teplica_poliv_message_PLC_M11 >2) THEN
						Modbus.Teplica_poliv_message_PLC	:=	11;
						Modbus.Teplica_poliv_status_PLC		:=	3;
					END_IF


			END_IF

			MB3.ReadRegs(Execute:= FALSE);
			state:=10;
		END_IF

10:
	IF (MBdataDO_byte <> MBdataDO_byte_old OR 	Cnt_Teplica_poliv_message_PLC_M9	>	0) THEN
	MB3.WriteMultipleCoils(
			UnitID:= teplica_ADM4188_id,
			Quantity:= 8,
			MBAddr:= 0,
			cbLength:= 16,
			pMemoryAddr:= ADR(MBdataDO_byte),
			Execute:= TRUE,
			Timeout:= T#2000ms,
			Busy => busy,
		);
		IF NOT busy THEN
			IF (mb3.Error = FALSE ) THEN
					Modbus.Teplica_poliv_message_PLC	:=	8;
					Cnt_Teplica_poliv_message_PLC_M9	 :=	0;


					IF (MBdataDO_byte.4=0 AND FertA_init_stop = TRUE) THEN
						Modbus.Cnt_water_fertA	:=	Modbus.Teplica_DI1_poliv -Cnt_water_fertA_start;
						Modbus.Teplica_time_elapsed_fertA :=(TIME_TO_UDINT( TIME() - t_Started_fertA))/1000;
						FertA_init_stop	:=	FALSE;
					END_IF

					IF (MBdataDO_byte.5=0 AND  FertB_init_stop = TRUE) THEN
						Modbus.Cnt_water_fertB	:=	Modbus.Teplica_DI1_poliv -Cnt_water_fertB_start;
						Modbus.Teplica_time_elapsed_fertB :=(TIME_TO_UDINT( TIME() - t_Started_fertB))/1000;
						FertB_init_stop	:=	FALSE;
					END_IF

					IF (  Poliv_init_stop = TRUE) THEN
						Modbus.Teplica_poliv_status_PLC :=  10;
						Poliv_init_stop := FALSE;
					END_IF


					MBdataDO_byte_old	:=	MBdataDO_byte;
			END_IF
			IF (mb3.Error = TRUE ) THEN

					Cnt_Teplica_poliv_message_PLC_M9	 :=	Cnt_Teplica_poliv_message_PLC_M9+1;
					IF (Cnt_Teplica_poliv_message_PLC_M9 >2) THEN
						Modbus.Teplica_poliv_message_PLC	:=	9;
						Modbus.Teplica_poliv_status_PLC	:=	3;
					END_IF

			END_IF



			MB3.ReadRegs(Execute:= FALSE);
			state:=15;

		END_IF
	ELSE

			IF (  Poliv_init_stop = TRUE) THEN
						Modbus.Teplica_poliv_status_PLC :=  10;
						Poliv_init_stop := FALSE;
			END_IF
			state:=15;

	END_IF




















15:

		MB3.ReadRegs(
			UnitID:= teplica_DS18B20_id,
			Quantity:= 8,
			MBAddr:= 0,
			cbLength:= 16,
			pMemoryAddr:= ADR(MBdata8),
			Execute:= TRUE,
			Timeout:=  T#2000ms,
			Busy => busy,
		);
		IF NOT busy THEN
			IF (mb3.Error = FALSE ) THEN
				IF (MBdata8[1] < 10000)
					THEN	teplica_DS18B20_temp[1]:=UINT_TO_REAL(MBdata8[1])/10;
				ELSE
					teplica_DS18B20_temp[1]:=-1*UINT_TO_REAL(MBdata8[1]-10000)/10;
				END_IF

				IF (MBdata8[2] < 10000)
					THEN	teplica_DS18B20_temp[2]:=UINT_TO_REAL(MBdata8[2])/10;
				ELSE
					teplica_DS18B20_temp[2]:=-1*UINT_TO_REAL(MBdata8[2]-10000)/10;
				END_IF


				IF (MBdata8[3] < 10000)
					THEN	teplica_DS18B20_temp[3]:=UINT_TO_REAL(MBdata8[3])/10;
				ELSE
					teplica_DS18B20_temp[3]:=-1*UINT_TO_REAL(MBdata8[3]-10000)/10;
				END_IF

				IF (MBdata8[4] < 10000)
					THEN	teplica_DS18B20_temp[4]:=UINT_TO_REAL(MBdata8[4])/10;
				ELSE
					teplica_DS18B20_temp[4]:=-1*UINT_TO_REAL(MBdata8[4]-10000)/10;
				END_IF

				Modbus.Teplica_temp_air			:=	teplica_DS18B20_temp[1];
				Modbus.Teplica_temp_ground		:=	teplica_DS18B20_temp[2];
				Modbus.Teplica_temp_pipe_heat 	:=	teplica_DS18B20_temp[3];
				Modbus.Teplica_temp_water_tank 	:=	teplica_DS18B20_temp[4];

			END_IF
			MB3.ReadRegs(Execute:= FALSE);
			state:=16;

		END_IF


16:

		MB3.ReadRegs(
			UnitID:= teplica_light_sensor_id,
			Quantity:= 2,
			MBAddr:= 2,
			cbLength:= 4,
			pMemoryAddr:= ADR(teplica_light_array),
			Execute:= TRUE,
			Timeout:= timeoutvalue,
			Busy => busy,
		);
		IF NOT busy THEN
			IF (mb3.Error = FALSE ) THEN
				teplica_light_high:=teplica_light_array[1];
				teplica_light_low:=teplica_light_array[2];
				teplica_light_dword:=(teplica_light_array[1]*65535)+teplica_light_array[2];

				Modbus.Teplica_light_lux		:=	DWORD_TO_REAL(teplica_light_dword);


			END_IF
			MB3.ReadRegs(Execute:= FALSE);
			state:=17;

		END_IF



17:

		MB3.ReadRegs(
			UnitID:= balkon_light_sensor_id,
			Quantity:= 1,
			MBAddr:= 6,
			cbLength:= 2,
			pMemoryAddr:= ADR(balkon_light_array),
			Execute:= TRUE,
			Timeout:= timeoutvalue,
			Busy => busy,
		);
		IF NOT busy THEN
			IF (mb3.Error = FALSE ) THEN
				balkon_light_high:=balkon_light_array[1];
				balkon_light_low:=balkon_light_array[2];
				balkon_light_word:=(balkon_light_array[2]*256)+balkon_light_array[1];

				Modbus.Balkon_light_lux		:=	WORD_TO_UDINT(balkon_light_word);
			END_IF
			MB3.ReadRegs(Execute:= FALSE);
			state:=18;

		END_IF


18:
		MB3.ReadRegs(
			UnitID:= sensors_SHT30_v3_id,
			Quantity:= 2,
			MBAddr:= 512,
			cbLength:= 6,
			pMemoryAddr:= ADR(MBdata),
			Execute:= TRUE,
			Timeout:= timeoutvalue,
			Busy => busy,
		);
		IF NOT busy THEN
			IF (mb3.Error = FALSE ) THEN
				sensors_SHT30_v3_temp:=INT_TO_REAL(MBdata[1])/10;
				sensors_SHT30_v3_hum:=INT_TO_REAL(MBdata[2])/10;

				Internal.Teplica_temp_SHT30		:=	sensors_SHT30_v3_temp;
				Internal.Teplica_hum_SHT30		:=	sensors_SHT30_v3_hum;
				Modbus.Teplica_temp_SHT30		:=	sensors_SHT30_v3_temp;
				Modbus.Teplica_hum_SHT30		:=	sensors_SHT30_v3_hum;
			END_IF
			MB3.ReadRegs(Execute:= FALSE);
			state :=19;
		END_IF

19:

		MB3.ReadRegs(
			UnitID:= sensor_teplica_PH_id,
			Quantity:= 1,
			MBAddr:= 0,
			cbLength:= 2,
			pMemoryAddr:= ADR(sensor_teplica_PH_int),
			Execute:= TRUE,
			Timeout:= timeoutvalue,
			Busy => busy,
		);
		IF NOT busy THEN
			IF (mb3.Error = FALSE ) THEN

				Modbus.Teplica_sensor_soil_PH		:=	INT_TO_REAL(sensor_teplica_PH_int)/100;
			END_IF
			MB3.ReadRegs(Execute:= FALSE);
			state:=20;

		END_IF

20:

		MB3.ReadRegs(
			UnitID:= sensor_teplica_EC_id,
			Quantity:= 4,
			MBAddr:= 0,
			cbLength:= 8,
			pMemoryAddr:= ADR(MBdata_sensor_teplica_EC),
			Execute:= TRUE,
			Timeout:= timeoutvalue,
			Busy => busy,
		);
		IF NOT busy THEN
			IF (mb3.Error = FALSE ) THEN
			Modbus.Teplica_sensor_soil_Hum	:=	INT_TO_REAL(MBdata_sensor_teplica_EC[1])/10;
			Modbus.Teplica_sensor_soil_Temp	:=	INT_TO_REAL(MBdata_sensor_teplica_EC[2])/10;
			Modbus.Teplica_sensor_soil_EC	:=	INT_TO_REAL(MBdata_sensor_teplica_EC[3]);
			Modbus.Teplica_sensor_soil_PH2	:=	INT_TO_REAL(MBdata_sensor_teplica_EC[4])/10;

			END_IF
			MB3.ReadRegs(Execute:= FALSE);
			state:=888;

		END_IF


888:
		TimerRS485_3(IN:=NOT TimerRS485_3Q , PT:=tTimerValue , Q=>TimerRS485_3Q , ET=> );
		IF TimerRS485_3.q THEN
			state:=0;
		END_IF


END_CASE

FtrigBusy(CLK:=mb3.BUSY );
IF FtrigBusy.Q THEN
	IF mb3.Error THEN
		LastModbusError := mb3.ErrorDiagnostics;
		LastErrorstate := state;
		CounterError := CounterError + 1;
	ELSE
		CounterSuccess := CounterSuccess + 1;
	END_IF
END_IF



SerialLinecontrolCom3(
	mode:=SerialLinemode_kl6_22b_standard,
	pComIn:=ADR(RS485read_3.MB3.InData),
	pComOut:=ADR(RS485read_3.MB3.OutData),
	SizeComIn:=SIZEOF(RS485read_3.MB3.OutData),
	TxBuffer:=TxBufferCom3,
	RxBuffer:=RxBufferCom3,
	Error=>,
	errorid=>);
END_PROGRAM

(* POU RS485read_3_old2, ST *)
PROGRAM RS485read_3_old2
VAR
(*	Period_vent_switch	: INT:=180; *)

	tTimerValue			: TIME	:=	t#3s; (* Период опроса RS485*)

(*	password_1				: ARRAY [1..6] OF BYTE:=6(1); (* пароль к меркуриям, по умолчанию 6 единиц*)
	crctest					: WORD;
	arrReceive				: ARRAY[1..22] OF BYTE;
	arrSend					: ARRAY[1..22] OF BYTE;
*)
	MBdata					 : ARRAY [1..2] OF INT;
	FtrigBusy				: F_TRIG;
	timeoutvalue				: TIME := T#1000ms;		(* timeout while waiting for an answer of the modbus slave *)
	state					: INT;
	busy					: BOOL;
	LastErrorstate				: INT;
	LastModbusError			: ST_ModbusErrorDiagnostics;
	CounterError				: DINT;
	CounterSuccess			: DINT;
	CounterError_M			: DINT;
	CounterSuccess_M		: DINT;

(*	i,k,l,m,t					: INT:=1; *)


	PWM_YC110_id			: BYTE:= 16#20 ; (*32 *)
	PWM_levels				 : ARRAY [1..4] OF INT;	(* reg dec 32*)
	PWM_levels_mem		 : ARRAY [1..4] OF INT;
	PWM_freq				 : ARRAY [1..4] OF INT; (* reg dec 64*)
	PWM_freq_mem			 : ARRAY [1..4] OF INT;
	PWM_cycle				 : ARRAY [1..4] OF INT;

	PWM_param_polar		:  INT;	(* reg dec 18*)
	PWM_param_polar_1		:  INT:=1;
	PWM_param_prz			: INT;	(* reg dec 30*)
	PWM_param_prz_1		: INT:=1;	(* reg dec 30*)

	PWM_cycle_1			:  UINT:=65535;
	PWM_cycle_2			:  UINT:=65535;
	PWM_cycle_3			:  UINT:=65535;
	PWM_cycle_4			:  UINT:=65535;

	teplica_DS18B20_id			: BYTE:=16#44;
	teplica_DS18B20_temp		: ARRAY[1..8] OF REAL:=8(0);
	MBdata8					 : ARRAY [1..8] OF UINT;

(*	Modbus_DO					: INT:=1; *)
	teplica_ADM4188_id			: BYTE:=16#45;
(*	teplica_ADM4188_DI_1			:  INT;
	teplica_ADM4188_DO_1		:  INT;
	teplica_ADM4188_DO_1_ACK	:  INT; *)

	teplica_light_sensor_id			: BYTE:=16#3C;
	teplica_light_low				: WORD;
	teplica_light_high				: WORD;
	teplica_light_dword				:DWORD;
	teplica_light_array				: ARRAY [1..2] OF WORD;








	MBdataDI		 			 : ARRAY [1..8] OF UINT;
	MBdataDO_byte					: INT;
	MBdataDO_byte_old				: INT;


(*	teplica_ADM4188_DO_ACK		:  INT;
	teplica_ADM4188_DI_ACK		: INT; *)
(*	teplica_ADM4188_DO_1		:  INT; *)

	zero						: INT:=0;



(*	TRIG_start_reset			:	R_TRIG; *)

	Teplica_DI1_cnt			:	UINT;
	Teplica_DI2_cnt			:	UINT;
	Teplica_DI3_cnt			:	UINT;
	Teplica_DI1_cnt_mem		:	UINT;
	Teplica_DI2_cnt_mem		:	UINT;
	Teplica_DI3_cnt_mem		:	UINT;

	check0					: INT:=0;
	check1					: INT:=0;
	check2					: INT:=0;
	check3					: INT:=0;

	sensors_SHT30_v3_id			:  BYTE:= 16#32 ;
	sensors_SHT30_v3_hum		:  REAL;
	sensors_SHT30_v3_temp		:  REAL;

	sensor_teplica_PH_id		: BYTE:= 16#78 ;
	sensor_teplica_PH_int		:INT;


	sensor_teplica_EC_id			: BYTE:= 16#C8 ;
	MBdata_sensor_teplica_EC		 : ARRAY [1..4] OF INT;

	cnt_clear_di_1			: BOOL;
	cnt_clear_di_2			: BOOL;
	cnt_clear_di_3			: BOOL;
	cnt_overload_1			:INT;
	cnt_overload_2			:INT;
	cnt_overload_3			:INT;
	password_1				: ARRAY [1..6] OF BYTE:=6(1); (* пароль к меркуриям, по умолчанию 6 единиц*)
	crctest					: WORD;
	get_energy_E_T1			: FB_GET_ENERGY;
	get_energy_E_T2			: FB_GET_ENERGY;
	get_energy_MT			: FB_GET_ENERGY;
	get_supply				: FB_GET_SUPPLY;
	get_current				: FB_GET_CURRENT;
	get_power				: FB_GET_POWER;
	energyMT					: ARRAY[1..12,1..2] OF REAL;

	get_current_done			: BOOL;
	get_power_done			: BOOL;

	get_energy_E_T1_done	: BOOL;
	get_energy_E_T2_done	: BOOL;
	get_energy_MT_done		: BOOL;

	get_supply_done			: BOOL;
	arrReceive				: ARRAY[1..5] OF BYTE;
	arrSend					: ARRAY[1..5] OF BYTE;
	i,k,l,m,t					: INT:=1;
	MBdata_sensor_ponics_PH : ARRAY [1..4] OF INT;
	Teplica_ph_sensor_temp	: REAL;

END_VAR
Modbus.RS485_3_cnt_error		:= CounterError;
Modbus.RS485_3_cnt_success	:= CounterSuccess;





CASE state OF
0:
	MB3.ReadRegs(Execute:= FALSE);
	state :=2;


2:
	MB3.WriteSingleRegister(
					UnitID:= PWM_YC110_id, (* station address *)
					Quantity:= 1,
					MBAddr:= 32,
					cbLength:= 2,
					pMemoryAddr:= ADR(fert_pwm_levelA),
					Execute:= TRUE,
					Timeout:= T#1000ms,
					Busy => busy,
					);
		IF NOT busy THEN
		(*	IF (mb3.Error = FALSE ) THEN

			END_IF
		*)
			MB3.ReadRegs(Execute:= FALSE);
			state:=3;
		END_IF

3:
	MB3.WriteSingleRegister(
					UnitID:= PWM_YC110_id, (* station address *)
					Quantity:= 1,
					MBAddr:= 33,
					cbLength:= 2,
					pMemoryAddr:= ADR(fert_pwm_levelB),
					Execute:= TRUE,
					Timeout:= T#1000ms,
					Busy => busy,
					);
		IF NOT busy THEN
		(*	IF (mb3.Error = FALSE ) THEN

			END_IF
		*)
			MB3.ReadRegs(Execute:= FALSE);
			state:=5;
		END_IF






4:
	MB3.WriteSingleRegister(
					UnitID:= PWM_YC110_id, (* station address *)
					Quantity:= 1,
					MBAddr:= 30,
					cbLength:= 2,
					pMemoryAddr:=ADR(PWM_param_prz_1) ,
					Execute:= TRUE,
					Timeout:= T#1000ms,
					Busy => busy,
					);
		IF NOT busy THEN
		(*	IF (mb3.Error = FALSE ) THEN

			END_IF
		*)
			MB3.ReadRegs(Execute:= FALSE);
			state:=5;
		END_IF


5:
	MB3.ReadRegs(
					UnitID:= PWM_YC110_id, (* station address *)
					Quantity:= 1,
					MBAddr:= 30,
					cbLength:= 2,
					pMemoryAddr:= ADR(PWM_param_prz),
					Execute:= TRUE,
					Timeout:= T#1000ms,
					Busy => busy,
					);
		IF NOT busy THEN
		(*	IF (mb3.Error = FALSE ) THEN

			END_IF
		*)
			MB3.ReadRegs(Execute:= FALSE);
			state:=10;
		END_IF



(*
6:
	MB3.WriteSingleRegister(
					UnitID:= PWM_YC110_id, (* station address *)
					Quantity:= 1,
					MBAddr:= 96,
					cbLength:= 2,
					pMemoryAddr:=ADR(PWM_cycle_1) ,
					Execute:= TRUE,
					Timeout:= T#1000ms,
					Busy => busy,
					);
		IF NOT busy THEN
		(*	IF (mb3.Error = FALSE ) THEN

			END_IF
		*)
			MB3.ReadRegs(Execute:= FALSE);
			state:=7;
		END_IF


7:
	MB3.WriteSingleRegister(
					UnitID:= PWM_YC110_id, (* station address *)
					Quantity:= 1,
					MBAddr:= 97,
					cbLength:= 2,
					pMemoryAddr:=ADR(PWM_cycle_2) ,
					Execute:= TRUE,
					Timeout:= T#1000ms,
					Busy => busy,
					);
		IF NOT busy THEN
		(*	IF (mb3.Error = FALSE ) THEN

			END_IF
		*)
			MB3.ReadRegs(Execute:= FALSE);
			state:=8;
		END_IF


8:
	MB3.WriteSingleRegister(
					UnitID:= PWM_YC110_id, (* station address *)
					Quantity:= 1,
					MBAddr:= 98,
					cbLength:= 2,
					pMemoryAddr:=ADR(PWM_cycle_3) ,
					Execute:= TRUE,
					Timeout:= T#1000ms,
					Busy => busy,
					);
		IF NOT busy THEN
		(*	IF (mb3.Error = FALSE ) THEN

			END_IF
		*)
			MB3.ReadRegs(Execute:= FALSE);
			state:=9;
		END_IF

9:
	MB3.WriteSingleRegister(
					UnitID:= PWM_YC110_id, (* station address *)
					Quantity:= 1,
					MBAddr:= 99,
					cbLength:= 2,
					pMemoryAddr:=ADR(PWM_cycle_4) ,
					Execute:= TRUE,
					Timeout:= T#1000ms,
					Busy => busy,
					);
		IF NOT busy THEN
		(*	IF (mb3.Error = FALSE ) THEN

			END_IF
		*)
			MB3.ReadRegs(Execute:= FALSE);
			state:=10;
		END_IF



*)


10:
	MB3.ReadRegs(
					UnitID:= PWM_YC110_id, (* station address *)
					Quantity:= 1,
					MBAddr:= 18,
					cbLength:= 2,
					pMemoryAddr:= ADR(PWM_param_polar),
					Execute:= TRUE,
					Timeout:= T#1000ms,
					Busy => busy,
					);
		IF NOT busy THEN
		(*	IF (mb3.Error = FALSE ) THEN

			END_IF
		*)
			MB3.ReadRegs(Execute:= FALSE);
			state:=11;
		END_IF

11:
	MB3.ReadRegs(
					UnitID:= PWM_YC110_id, (* station address *)
					Quantity:= 4,
					MBAddr:= 96,
					cbLength:= 8,
					pMemoryAddr:= ADR(PWM_cycle),
					Execute:= TRUE,
					Timeout:= T#1000ms,
					Busy => busy,
					);
		IF NOT busy THEN
		(*	IF (mb3.Error = FALSE ) THEN

			END_IF
		*)
			MB3.ReadRegs(Execute:= FALSE);
			state:=13;
		END_IF



13:
	MB3.ReadRegs(
					UnitID:= PWM_YC110_id, (* station address *)
					Quantity:= 4,
					MBAddr:= 32,
					cbLength:= 8,
					pMemoryAddr:= ADR(PWM_levels),
					Execute:= TRUE,
					Timeout:= T#1000ms,
					Busy => busy,
					);
		IF NOT busy THEN
			IF (mb3.Error = FALSE ) THEN
				PWM_levels_mem[1]	:=	PWM_levels[1];
				PWM_levels_mem[2]	:=	PWM_levels[2];
				PWM_levels_mem[3]	:=	PWM_levels[3];
				PWM_levels_mem[4]	:=	PWM_levels[4];

			END_IF

			MB3.ReadRegs(Execute:= FALSE);
			state:=14;
		END_IF

14:
	MB3.ReadRegs(
					UnitID:= PWM_YC110_id, (* station address *)
					Quantity:= 4,
					MBAddr:= 64,
					cbLength:= 8,
					pMemoryAddr:= ADR(PWM_freq),
					Execute:= TRUE,
					Timeout:= T#1000ms,
					Busy => busy,
					);
		IF NOT busy THEN
			IF (mb3.Error = FALSE ) THEN
				PWM_freq_mem[1]	:=	PWM_freq[1];
				PWM_freq_mem[2]	:=	PWM_freq[2];
				PWM_freq_mem[3]	:=	PWM_freq[3];
				PWM_freq_mem[4]	:=	PWM_freq[4];

			END_IF

			MB3.ReadRegs(Execute:= FALSE);
			state:=15;
		END_IF


15:

		MB3.ReadRegs(
			UnitID:= teplica_DS18B20_id,
			Quantity:= 8,
			MBAddr:= 0,
			cbLength:= 16,
			pMemoryAddr:= ADR(MBdata8),
			Execute:= TRUE,
			Timeout:=  T#2000ms,
			Busy => busy,
		);
		IF NOT busy THEN
			IF (mb3.Error = FALSE ) THEN
				IF (MBdata8[1] < 10000)
					THEN	teplica_DS18B20_temp[1]:=UINT_TO_REAL(MBdata8[1])/10;
				ELSE
					teplica_DS18B20_temp[1]:=-1*UINT_TO_REAL(MBdata8[1]-10000)/10;
				END_IF

				IF (MBdata8[2] < 10000)
					THEN	teplica_DS18B20_temp[2]:=UINT_TO_REAL(MBdata8[2])/10;
				ELSE
					teplica_DS18B20_temp[2]:=-1*UINT_TO_REAL(MBdata8[2]-10000)/10;
				END_IF


				IF (MBdata8[3] < 10000)
					THEN	teplica_DS18B20_temp[3]:=UINT_TO_REAL(MBdata8[3])/10;
				ELSE
					teplica_DS18B20_temp[3]:=-1*UINT_TO_REAL(MBdata8[3]-10000)/10;
				END_IF

				IF (MBdata8[4] < 10000)
					THEN	teplica_DS18B20_temp[4]:=UINT_TO_REAL(MBdata8[4])/10;
				ELSE
					teplica_DS18B20_temp[4]:=-1*UINT_TO_REAL(MBdata8[4]-10000)/10;
				END_IF

				IF  (teplica_DS18B20_temp[1] <>0 AND teplica_DS18B20_temp[1] <>85)	THEN
					Modbus.Teplica_temp_air			:=	teplica_DS18B20_temp[1];
				END_IF

				IF  (teplica_DS18B20_temp[2] <>0 AND teplica_DS18B20_temp[2] <>85)	THEN
					Modbus.Teplica_temp_ground		:=	teplica_DS18B20_temp[2];
				END_IF

				IF  (teplica_DS18B20_temp[3] <>0 AND teplica_DS18B20_temp[3] <>85)	THEN
					Modbus.Teplica_temp_pipe_heat 	:=	teplica_DS18B20_temp[3];
				END_IF

				IF  (teplica_DS18B20_temp[4] <>0 AND teplica_DS18B20_temp[4] <>85)	THEN
					Modbus.Teplica_temp_water_tank 	:=	teplica_DS18B20_temp[4];
				END_IF


			END_IF
			MB3.ReadRegs(Execute:= FALSE);
			state:=16;

		END_IF


16:

		MB3.ReadRegs(
			UnitID:= teplica_light_sensor_id,
			Quantity:= 2,
			MBAddr:= 2,
			cbLength:= 4,
			pMemoryAddr:= ADR(teplica_light_array),
			Execute:= TRUE,
			Timeout:= timeoutvalue,
			Busy => busy,
		);
		IF NOT busy THEN
			IF (mb3.Error = FALSE ) THEN
				teplica_light_high:=teplica_light_array[1];
				teplica_light_low:=teplica_light_array[2];
				teplica_light_dword:=(teplica_light_array[1]*65535)+teplica_light_array[2];

				Modbus.Teplica_light_lux		:=	DWORD_TO_REAL(teplica_light_dword);


			END_IF
			MB3.ReadRegs(Execute:= FALSE);
			state:=18;

		END_IF





18:
		MB3.ReadRegs(
			UnitID:= sensors_SHT30_v3_id,
			Quantity:= 2,
			MBAddr:= 512,
			cbLength:= 6,
			pMemoryAddr:= ADR(MBdata),
			Execute:= TRUE,
			Timeout:= timeoutvalue,
			Busy => busy,
		);
		IF NOT busy THEN
			IF (mb3.Error = FALSE ) THEN
				sensors_SHT30_v3_temp:=INT_TO_REAL(MBdata[1])/10;
				sensors_SHT30_v3_hum:=INT_TO_REAL(MBdata[2])/10;

				Internal.Teplica_temp_SHT30		:=	sensors_SHT30_v3_temp;
				Internal.Teplica_hum_SHT30		:=	sensors_SHT30_v3_hum;
				Modbus.Teplica_temp_SHT30		:=	sensors_SHT30_v3_temp;
				Modbus.Teplica_hum_SHT30		:=	sensors_SHT30_v3_hum;
			END_IF
			MB3.ReadRegs(Execute:= FALSE);
			state :=19;
		END_IF

19:

		MB3.ReadRegs(
			UnitID:= sensor_teplica_PH_id,
			(*Quantity:= 1,
			MBAddr:= 0,
			cbLength:= 2,
			pMemoryAddr:= ADR(sensor_teplica_PH_int),*)
			Quantity:= 4,
			MBAddr:= 0,
			cbLength:= 8,
			pMemoryAddr:= ADR(MBdata_sensor_ponics_PH),
			Execute:= TRUE,
			Timeout:= timeoutvalue,
			Busy => busy,
		);
		IF NOT busy THEN
			IF (mb3.Error = FALSE ) THEN

(*				Modbus.Teplica_sensor_soil_PH		:=	INT_TO_REAL(sensor_teplica_PH_int)/100;	*)
				Modbus.Teplica_sensor_soil_PH	:=	INT_TO_REAL(MBdata_sensor_ponics_PH[1])/100;
				Teplica_ph_sensor_temp			:=	INT_TO_REAL(MBdata_sensor_ponics_PH[3])/10;

			END_IF
			MB3.ReadRegs(Execute:= FALSE);
			state:=20;

		END_IF

20:

		MB3.ReadRegs(
			UnitID:= sensor_teplica_EC_id,
			Quantity:= 4,
			MBAddr:= 0,
			cbLength:= 8,
			pMemoryAddr:= ADR(MBdata_sensor_teplica_EC),
			Execute:= TRUE,
			Timeout:= timeoutvalue,
			Busy => busy,
		);
		IF NOT busy THEN
			IF (mb3.Error = FALSE ) THEN
			Modbus.Teplica_sensor_soil_Hum	:=	INT_TO_REAL(MBdata_sensor_teplica_EC[1])/10;
			Modbus.Teplica_sensor_soil_Temp	:=	INT_TO_REAL(MBdata_sensor_teplica_EC[2])/10;
			Modbus.Teplica_sensor_soil_EC	:=	INT_TO_REAL(MBdata_sensor_teplica_EC[3]);
			Modbus.Teplica_sensor_soil_PH2	:=	INT_TO_REAL(MBdata_sensor_teplica_EC[4])/10;

			END_IF
			MB3.ReadRegs(Execute:= FALSE);
			state:=105;

		END_IF



(*	state:=105; *)

105: (*открываем канал*)


	Clear(Buffer := RxBufferCom3);
	arrSend[1]:=Merc_address;
	arrSend[2]:=1; (*код доступа*)
	arrSend[3]:=1; (*Уровень доступа*)

	MEMCPY(ADR(arrSend)+3,ADR(password_1),6); (*пароль*)
	crctest:=F_CRC16(ADR(arrSend),9); (*расчет контрольной суммы*)
	MEMCPY(ADR(arrSend)+9,ADR(crctest),SIZEOF(crctest)); (*прибавление контрольной суммы к запросу*)
	SendDataCom3(pSendData:=ADR(arrSend),Length:=11,TXBuffer:=TxBufferCom3,Busy=>,Error=>);
(*	tmCheck(in:=FALSE); *)
	tmCheckM(in:=FALSE);
	tmCheckM(in:=TRUE, pt:=t#3s); 	(*запуск таймера проверки - потеря связи\обрыв кабеля*)
	state:=106;

106: (*ответ*)
	ReceiveDataCom3(pPrefix:=,LenPrefix:=,pSuffix:=,LenSuffix:=,
	pReceiveData:=ADR(arrReceive),SizeReceiveData:=4,
	Timeout:=t#2s,Reset:=,
	RXbuffer:=RxBufferCom3,
	DataReceived=>,busy=>,Error=>,RxTimeout=>,LenReceiveData=>);
	IF ReceiveDataCom3.Error <> 0 THEN
		state:=888;
	END_IF
	IF receiveDataCom3.DataReceived THEN
		state:=107;
	ELSIF tmCheckM.Q THEN
		state:=888;
	END_IF
107: (*проверка ответа*)

	IF arrReceive[1] = Merc_address THEN
		state:= 108;
	ELSE
		state:=888;
	END_IF



108:
	(*	tmCheck(in:=FALSE);	*)
		tmCheck(in:=NOT tmCheck.q,pt:=t#2s);
		get_supply_done := FALSE;
		get_supply( byte1:=16#8, byte2:=16#16, byte3:=16#11,  supply1=>Modbus.UV1,supply2=>Modbus.UV2,supply3=>Modbus.UV3, done=>get_supply_done);
		IF get_supply_done = TRUE THEN
			CounterSuccess := CounterSuccess+1;
			state:=109;
		ELSIF tmcheck.Q THEN
			CounterError := CounterError+1;
			 state:=888;
		END_IF



 (*запрос на чтение тока  на всех фазах
--------------------------------------------------------------------------------------------------------------------------------------------------------------------
*)
109:
	(*	tmCheck(in:=FALSE);	*)
		tmCheck(in:=NOT tmCheck.q,pt:=t#2s);
		get_current_done := FALSE;
		get_current(byte1:=16#8, byte2:=16#16, byte3:=16#21,  current1=>Modbus.Ia1,current2=>Modbus.Ia2,current3=>Modbus.Ia3, done=>get_current_done);
		IF get_current_done = TRUE THEN
			state:=110;
		ELSIF tmcheck.Q THEN state:=888;
		END_IF

 (*запрос на чтение мощности  на всех фазах
--------------------------------------------------------------------------------------------------------------------------------------------------------------------
*)

110:
	(*	tmCheck(in:=FALSE);	*)
		tmCheck(in:=NOT tmCheck.q,pt:=t#2s);
		get_power_done := FALSE;
		get_power(byte1:=16#8, byte2:=16#16, byte3:=16#0,  power_total=>Modbus.pw_total, power1=>Modbus.pw1, power2=>Modbus.pw2,power3=>Modbus.pw3,done=>get_power_done);
		IF get_power_done = TRUE THEN
			state:=111;
		ELSIF tmcheck.Q THEN state:=888;
		END_IF

 (*запрос на чтение энергии T1
--------------------------------------------------------------------------------------------------------------------------------------------------------------------
*)
111:
	(*	tmCheck(in:=FALSE);	*)
		tmCheck(in:=NOT tmCheck.q,pt:=t#2s);
		get_energy_E_T1_done := FALSE;
		get_energy_E_T1(byte1:=5, byte2:=16#0, byte3:=1,  energy=>Modbus.E_T1, done=>get_energy_E_T1_done);
		IF get_energy_E_T1_done = TRUE THEN
			state:=112;
		ELSIF tmcheck.Q THEN state:=888;
		END_IF
 (*запрос на чтение энергии T2
--------------------------------------------------------------------------------------------------------------------------------------------------------------------
*)

112:
	(*	tmCheck(in:=FALSE);	*)
		tmCheck(in:=NOT tmCheck.q,pt:=t#2s);
		get_energy_E_T2_done := FALSE;
		get_energy_E_T2(byte1:=5, byte2:=16#0, byte3:=2,  energy=>Modbus.E_T2, done=>get_energy_E_T2_done);
		IF get_energy_E_T2_done = TRUE THEN
			state:=888;
		ELSIF tmcheck.Q THEN state:=888;
		END_IF

113:
		Timer_day(IN:=NOT Timer_dayQ , PT:=T#30m , Q=>Timer_dayQ , ET=> );
			IF timer_day.q THEN
				state:=114;
			ELSE
				state:=888;
			END_IF

114:
	(*	tmCheck(in:=FALSE);	*)
		tmCheckE(in:=NOT tmCheckE.q,pt:=t#2s, Q=>tmCheckEQ , ET=>);
		get_energy_MT_done := FALSE;

	(*	IF (tmCheckEQ) THEN *)
			get_energy_MT(byte1:=5, byte2:=INT_TO_BYTE(48+m), byte3:=INT_TO_BYTE(t),   energy=>energyMT[m,t],done=>get_energy_MT_done);
(*		END_IF *)

		IF get_energy_MT_done = TRUE THEN
			t:=t+1;
			IF (t>2 AND m<13) THEN
				t:=1;
				m:=m+1;
				state:=114;
			END_IF

					IF ( m=13) THEN
						t:=1;
						m:=1;
						Modbus.M1T1:=energyMT[1,1];
						Modbus.M1T2:=energyMT[1,2];
						Modbus.M2T1:=energyMT[2,1];
						Modbus.M2T2:=energyMT[2,2];
						Modbus.M3T1:=energyMT[3,1];
						Modbus.M3T2:=energyMT[3,2];
						Modbus.M4T1:=energyMT[4,1];
						Modbus.M4T2:=energyMT[4,2];
						Modbus.M5T1:=energyMT[5,1];
						Modbus.M5T2:=energyMT[5,2];
						Modbus.M6T1:=energyMT[6,1];
						Modbus.M6T2:=energyMT[6,2];
						Modbus.M7T1:=energyMT[7,1];
						Modbus.M7T2:=energyMT[7,2];
						Modbus.M8T1:=energyMT[8,1];
						Modbus.M8T2:=energyMT[8,2];
						Modbus.M9T1:=energyMT[9,1];
						Modbus.M9T2:=energyMT[9,2];
						Modbus.M10T1:=energyMT[10,1];
						Modbus.M10T2:=energyMT[10,2];
						Modbus.M11T1:=energyMT[11,1];
						Modbus.M11T2:=energyMT[11,2];
						Modbus.M12T1:=energyMT[12,1];
						Modbus.M12T2:=energyMT[12,2];
						state:=888;
					END_IF
		ELSIF tmcheckE.Q THEN state:=114;
		END_IF






888:
		TimerRS485_3(IN:=NOT TimerRS485_3Q , PT:=tTimerValue , Q=>TimerRS485_3Q , ET=> );
		IF TimerRS485_3.q THEN
			state:=0;
		END_IF


END_CASE

FtrigBusy(CLK:=mb3.BUSY );
IF FtrigBusy.Q THEN
	IF mb3.Error THEN
		LastModbusError := mb3.ErrorDiagnostics;
		LastErrorstate := state;
		CounterError := CounterError + 1;
	ELSE
		CounterSuccess := CounterSuccess + 1;
	END_IF
END_IF



SerialLinecontrolCom3(
	mode:=SerialLinemode_kl6_22b_standard,
	pComIn:=ADR(RS485read_3.MB3.InData),
	pComOut:=ADR(RS485read_3.MB3.OutData),
	SizeComIn:=SIZEOF(RS485read_3.MB3.OutData),
	TxBuffer:=TxBufferCom3,
	RxBuffer:=RxBufferCom3,
	Error=>,
	errorid=>);
END_PROGRAM

(* POU Security, ST *)
PROGRAM Security
VAR
	TRIG_PIR_terrasa			:	F_TRIG;
	TRIG_PIR_zapad			:	F_TRIG;
	TRIG_PIR_vostok			:	F_TRIG;
	TRIG_PIR_sport			:	F_TRIG;
	TRIG_GERKON_drovnik	:	F_TRIG;
	TRIG_sensor_smoke_1floor:	F_TRIG;

	trig_mem_terrasa				:	BOOL:=FALSE;
	trig_mem_zapad				:	BOOL:=FALSE;
	trig_mem_vostok				:	BOOL:=FALSE;
	trig_mem_sport				:	BOOL:=FALSE;
	trig_mem_drovnik				:	BOOL:=FALSE;
	trig_mem_sensor_smoke_1floor	:	BOOL:=FALSE;

END_VAR
(*  Используем триггеры для исключения ложной информации о сработке датчиков при перезагрузке ПЛК *)


TRIG_PIR_terrasa(CLK :=HW_PIR_terrasa);
TRIG_PIR_zapad(CLK :=HW_PIR_zapad);
TRIG_PIR_vostok(CLK :=HW_PIR_vostok);
TRIG_PIR_sport(CLK :=HW_PIR_sport);
TRIG_GERKON_drovnik(CLK :=HW_GERKON_drovnik);
TRIG_sensor_smoke_1floor(CLK :=HW_sensor_smoke_1floor);


IF (NOT TRIG_PIR_terrasa.Q) THEN
	iobroker.PIR_terrasa:=NOT TRIG_PIR_terrasa.Q;
END_IF
IF (trig_mem_terrasa=TRUE) THEN
	iobroker.PIR_terrasa:=FALSE;
	trig_mem_terrasa:=FALSE;
END_IF
IF (TRIG_PIR_terrasa.Q) THEN
	trig_mem_terrasa:=TRUE;
END_IF



IF (NOT TRIG_PIR_zapad.Q) THEN
	iobroker.PIR_zapad:=NOT TRIG_PIR_zapad.Q;
END_IF
IF (trig_mem_zapad=TRUE) THEN
	iobroker.PIR_zapad:=FALSE;
	trig_mem_zapad:=FALSE;
END_IF
IF (TRIG_PIR_zapad.Q) THEN
	trig_mem_zapad:=TRUE;
END_IF


IF (NOT TRIG_PIR_vostok.Q) THEN
	iobroker.PIR_vostok:=NOT TRIG_PIR_vostok.Q;
END_IF
IF (trig_mem_vostok=TRUE) THEN
	iobroker.PIR_vostok:=FALSE;
	trig_mem_vostok:=FALSE;
END_IF
IF (TRIG_PIR_vostok.Q) THEN
	trig_mem_vostok:=TRUE;
END_IF


IF (NOT TRIG_PIR_sport.Q) THEN
	iobroker.PIR_sport:=NOT TRIG_PIR_sport.Q;
END_IF
IF (trig_mem_sport=TRUE) THEN
	iobroker.PIR_sport:=FALSE;
	trig_mem_sport:=FALSE;
END_IF
IF (TRIG_PIR_sport.Q) THEN
	trig_mem_sport:=TRUE;
END_IF

IF (NOT TRIG_GERKON_drovnik.Q) THEN
	iobroker.GERKON_drovnik:=NOT TRIG_GERKON_drovnik.Q;
END_IF
IF (trig_mem_drovnik=TRUE) THEN
	iobroker.GERKON_drovnik:=FALSE;
	trig_mem_drovnik:=FALSE;
END_IF
IF (TRIG_GERKON_drovnik.Q) THEN
	trig_mem_drovnik:=TRUE;
END_IF


IF (NOT TRIG_sensor_smoke_1floor.Q) THEN
	iobroker.SMOKE:=NOT TRIG_sensor_smoke_1floor.Q;
END_IF
IF (trig_mem_sensor_smoke_1floor=TRUE) THEN
	iobroker.SMOKE:=FALSE;
	trig_mem_sensor_smoke_1floor:=FALSE;
END_IF
IF (TRIG_sensor_smoke_1floor.Q) THEN
	trig_mem_sensor_smoke_1floor:=TRUE;
END_IF
END_PROGRAM

(* POU Teplica, ST *)
PROGRAM Teplica
VAR
	Timer_poliv_all			: TON;
	Timer_poliv_allQ			: BOOL;

	Timer_1_clear			: TON;
	Timer_2_fertA				: TON;
	Timer_3_clear			: TON;
	Timer_4_fertB				: TON;
	Timer_poliv_with_fert		: TON;

	Timer_1_clearQ			: BOOL;
	Timer_2_fertAQ			: BOOL;
	Timer_3_clearQ			: BOOL;
	Timer_4_fertBQ			: BOOL;
	Step_1_clear				: BOOL;

	 tTimerValue_poliv_all		: TIME:=t#60s;  (* Максимальное время полива*)
	 tTimerValue_1_clear		: TIME:=t#10s;  (* Промывка перед 1 фертигацией*)
	 tTimerValue_2_fertA		: TIME:=t#30s;  (* Ограничение фертигации из бака А*)
	 tTimerValue_3_clear		: TIME:=t#60s;  (* Промывка перед OFF*)
	 tTimerValue_4_fertB		: TIME:=t#10s;  (* Ограничение фертигации из бака Б*)
	 tTimerValue_poliv_with_fert	: TIME:=t#90m;  (* Ограничение полива с фертигацией *)

	Timer_valve				: TON;
	Timer_valveQ			: BOOL;
	 tTimerValue_valve_water	: TIME:=t#60m;  (* Максимальное время открытия клапана подачи воды в теплицу*)

	TRIG_start_poliv			:	R_TRIG;
	TRIG_valve_tank_F		:	F_TRIG;
	TRIG_valve_tank_R		:	R_TRIG;


(*	TRIG_end_poliv_timer		:	R_TRIG; *)
(*	TRIG_end_poliv_count		:	R_TRIG; *)

	Bool_poliv_before_fert		: 	BOOL;

	TRIG_poliv_break			:	R_TRIG;

(*	TRIG_end_1_clear_timer	:	R_TRIG; *)
(*	TRIG_end_1_clear_cnt		:	R_TRIG; *)
(*	TRIG_end_2_fertA_timer	:	R_TRIG; *)
(*	TRIG_end_2_fertA_cnt		:	R_TRIG; *)
(*	TRIG_end_3_clear_timer	:	R_TRIG; *)
(*	TRIG_end_3_clear_cnt		:	R_TRIG; *)
(*	TRIG_end_4_fertB_timer	:	R_TRIG; *)
(*	TRIG_end_4_fertB_cnt		:	R_TRIG; *)

(*	BOOL_cnt_poliv			:	BOOL;
	BOOL_cnt_fertA			:	BOOL;
	BOOL_cnt_fertB			:	BOOL; *)

	Poliv_liters				:	REAL;
	FertA_liters				:	REAL;
	FertB_liters				:	REAL;
(*
	Cnt_water_fertA_start		:	UDINT;
	Cnt_water_fertB_start		:	UDINT;
*)
(*
	t_Started_poliv			:	TIME;
	t_Started_fertA			:	TIME;
	t_Started_fertB			:	TIME;
*)
	gisterezis_lux				:	INT:=1000;
	Poliv_before_fert			:	INT:=0;
	Timer_poliv_with_fertQ		: 	BOOL;
	Trigger_water_impulse_teplica	: F_TRIG;
	Trigger_water_impulse2_teplica	: R_TRIG;

	Trigger_fertA_impulse_teplica	: F_TRIG;
	Trigger_fertB_impulse_teplica	: F_TRIG;

	Impulse_water_teplica		:	UDINT:=0;
	Impulse2_water_teplica	:	UDINT:=0;
	Impulse_fertA_teplica		:	UDINT:=0;
	Impulse_fertB_teplica		:	UDINT:=0;

END_VAR
Trigger_water_impulse_teplica(CLK:=HW_impulse_water_teplica);
Trigger_water_impulse2_teplica(CLK:=HW_impulse_water_teplica);

Trigger_fertA_impulse_teplica(CLK:=HW_impulse_fertA_teplica);
Trigger_fertB_impulse_teplica(CLK:=HW_impulse_fertB_teplica);

IF Trigger_water_impulse_teplica.Q THEN
	Impulse_water_teplica	:= 	Impulse_water_teplica+1;
END_IF
IF Trigger_water_impulse2_teplica.Q THEN
	Impulse2_water_teplica	:= 	Impulse2_water_teplica+1;
END_IF


IF Trigger_fertA_impulse_teplica.Q THEN
	Impulse_fertA_teplica	:= 	Impulse_fertA_teplica+1;
END_IF
IF Trigger_fertB_impulse_teplica.Q THEN
	Impulse_fertB_teplica	:= 	Impulse_fertB_teplica+1;
END_IF



tTimerValue_poliv_all	:=	UDINT_TO_TIME(60*1000*Modbus.Teplica_set_max_poliv_time);
tTimerValue_1_clear	:=	UDINT_TO_TIME(60*1000*Modbus.Teplica_set_clear_time);
tTimerValue_2_fertA	:=	UDINT_TO_TIME(60*1000*Modbus.Teplica_set_max_fertA_time);
tTimerValue_3_clear	:=	t#60s;
tTimerValue_4_fertB	:=	UDINT_TO_TIME(60*1000*Modbus.Teplica_set_max_fertB_time);



Timer_poliv_all();
Timer_poliv_with_fert();
Timer_1_clear();
Timer_2_fertA();
Timer_3_clear();
Timer_4_fertB();
Timer_valve();


TRIG_start_poliv(CLK :=Modbus.Teplica_poliv_active);
TRIG_poliv_break(CLK :=Modbus.Teplica_poliv_break);

TRIG_valve_tank_F(CLK:=HW_water_tank_teplica_level);
TRIG_valve_tank_R(CLK:=HW_water_tank_teplica_level);

Modbus.Teplica_tank_teplica_level	:=	HW_water_tank_teplica_level;

IF (TRIG_valve_tank_F.Q) THEN
	Timer_valve(IN:=NOT Timer_valveQ , PT:=tTimerValue_valve_water , Q=>Timer_valveQ , ET=> );
	HW_valve_pomp_teplica :=	TRUE;
END_IF

IF (TRIG_valve_tank_R.Q	OR Timer_valveQ = TRUE) THEN
	HW_valve_pomp_teplica :=	FALSE;
	Timer_valveQ	:= FALSE;
	Timer_valve.IN	:= FALSE;
END_IF



IF (TRIG_start_poliv.Q AND  Modbus.Teplica_poliv_status_PLC <> 2)   THEN
		Cnt_cleared	:= 	FALSE;
		Step_1_clear	 :=	FALSE;
		Poliv_liters	:=	0;
		FertA_liters	:=	0;
		FertB_liters	:=	0;
		Cnt_water_fertA_start	:=	0;
		Cnt_water_fertB_start	:=	0;
		Modbus.Cnt_water_fertA	:=	0;
		Modbus.Cnt_water_fertB	:=	0;
		Modbus.Teplica_DI1_poliv	:=	0;
		Modbus.Teplica_DI2_fertA	:=	0;
		Modbus.Teplica_DI3_fertB	:=	0;
		Modbus.Teplica_poliv_status_PLC:=1;
		Modbus.Teplica_poliv_message_PLC:=1;
		Modbus.Teplica_time_elapsed_poliv :=0;
		Modbus.Teplica_time_elapsed_fertA :=0;
		Modbus.Teplica_time_elapsed_fertB :=0;

		Timer_1_clearQ			:= FALSE;
		Timer_2_fertAQ			:= FALSE;
		Timer_3_clearQ			:= FALSE;
		Timer_4_fertBQ			:= FALSE;
		Step_1_clear				:= FALSE;
		Poliv_init_stop			:= FALSE;
		FertA_init_stop			:=	FALSE;
		FertB_init_stop			:=	FALSE;
		Bool_poliv_before_fert		:=	FALSE;
END_IF

